C03650=1184.713,-44.316,-42.579,179.626,5.711,149.123
C03651=1184.719,-44.566,-42.567,179.624,5.710,149.123
C03652=1184.724,-44.815,-42.555,179.621,5.710,149.124
C03653=1184.729,-45.065,-42.544,179.619,5.709,149.125
C03654=1184.734,-45.315,-42.532,179.617,5.709,149.125
C03655=1184.740,-45.564,-42.520,179.614,5.709,149.126
C03656=1184.745,-45.814,-42.509,179.612,5.708,149.127
C03657=1184.750,-46.063,-42.496,179.609,5.708,149.127
C03658=1184.755,-46.313,-42.484,179.607,5.708,149.128
C03659=1184.761,-46.563,-42.473,179.605,5.708,149.129
C03660=1184.766,-46.813,-42.461,179.602,5.707,149.129
C03661=1184.771,-47.063,-42.449,179.600,5.707,149.130
C03662=1184.776,-47.312,-42.437,179.598,5.707,149.130
C03663=1184.781,-47.561,-42.425,179.595,5.706,149.131
C03664=1184.786,-47.811,-42.414,179.592,5.706,149.132
C03665=1184.791,-48.061,-42.402,179.591,5.706,149.132
C03666=1184.797,-48.310,-42.391,179.588,5.705,149.133
C03667=1184.802,-48.560,-42.379,179.586,5.705,149.134
C03668=1184.807,-48.810,-42.368,179.583,5.704,149.134
C03669=1184.812,-49.060,-42.356,179.581,5.704,149.135
C03670=1184.818,-49.330,-42.343,179.579,5.704,149.136
C03671=1184.824,-49.600,-42.330,179.576,5.704,149.136
C03672=1184.829,-49.871,-42.318,179.573,5.703,149.137
C03673=1184.835,-50.141,-42.305,179.571,5.703,149.138
C03674=1184.841,-50.390,-42.293,179.568,5.702,149.138
C03675=1184.845,-50.640,-42.282,179.566,5.702,149.139
C03676=1184.851,-50.890,-42.270,179.564,5.702,149.140
C03677=1184.855,-51.140,-42.259,179.561,5.701,149.140
C03678=1184.861,-51.389,-42.247,179.559,5.701,149.141
C03679=1184.866,-51.639,-42.235,179.557,5.701,149.142
C03680=1184.871,-51.889,-42.224,179.554,5.701,149.142
C03681=1184.877,-52.138,-42.212,179.552,5.700,149.143
C03682=1184.882,-52.388,-42.201,179.550,5.700,149.143
C03683=1184.887,-52.638,-42.189,179.547,5.700,149.144
C03684=1184.892,-52.887,-42.178,179.544,5.699,149.145
C03685=1184.897,-53.137,-42.166,179.542,5.698,149.145
C03686=1184.903,-53.386,-42.155,179.540,5.699,149.146
C03687=1184.908,-53.636,-42.143,179.538,5.698,149.147
C03688=1184.913,-53.886,-42.132,179.535,5.698,149.147
C03689=1184.918,-54.136,-42.120,179.533,5.697,149.148
C03690=1184.923,-54.385,-42.109,179.531,5.698,149.149
C03691=1184.928,-54.635,-42.097,179.528,5.697,149.149
C03692=1184.934,-54.884,-42.086,179.526,5.696,149.150
C03693=1184.939,-55.134,-42.074,179.524,5.697,149.150
C03694=1184.944,-55.384,-42.063,179.521,5.696,149.151
C03695=1184.949,-55.634,-42.051,179.519,5.695,149.152
C03696=1184.954,-55.883,-42.040,179.516,5.695,149.152
C03697=1184.960,-56.133,-42.028,179.514,5.695,149.153
C03698=1184.965,-56.382,-42.017,179.512,5.695,149.154
C03699=1184.970,-56.633,-42.006,179.509,5.694,149.154
C03700=1184.975,-56.882,-41.994,179.507,5.694,149.155
C03701=1184.981,-57.132,-41.983,179.505,5.694,149.155
C03702=1184.986,-57.381,-41.971,179.502,5.693,149.156
C03703=1184.990,-57.631,-41.960,179.500,5.694,149.157
C03704=1184.996,-57.881,-41.948,179.498,5.693,149.158
C03705=1185.001,-58.130,-41.937,179.495,5.692,149.158
C03706=1185.007,-58.380,-41.926,179.493,5.692,149.159
C03707=1185.012,-58.630,-41.915,179.491,5.692,149.159
C03708=1185.016,-58.880,-41.904,179.488,5.691,149.160
C03709=1185.022,-59.129,-41.892,179.486,5.691,149.161
C03710=1185.027,-59.378,-41.881,179.484,5.691,149.161
C03711=1185.033,-59.629,-41.870,179.482,5.691,149.162
C03712=1185.037,-59.879,-41.858,179.479,5.690,149.162
C03713=1185.043,-60.128,-41.847,179.477,5.691,149.163
C03714=1185.048,-60.378,-41.836,179.475,5.690,149.164
C03715=1185.053,-60.628,-41.825,179.472,5.689,149.164
C03716=1185.058,-60.878,-41.813,179.470,5.690,149.165
C03717=1185.064,-61.127,-41.802,179.467,5.689,149.166
C03718=1185.068,-61.376,-41.791,179.465,5.688,149.166
C03719=1185.074,-61.627,-41.780,179.462,5.688,149.167
C03720=1185.080,-61.876,-41.769,179.460,5.688,149.168
C03721=1185.084,-62.125,-41.757,179.458,5.688,149.168
C03722=1185.090,-62.375,-41.746,179.455,5.687,149.169
C03723=1185.095,-62.625,-41.735,179.453,5.688,149.170
C03724=1185.100,-62.874,-41.724,179.451,5.687,149.170
C03725=1185.105,-63.124,-41.712,179.448,5.686,149.171
C03726=1185.110,-63.375,-41.702,179.446,5.687,149.171
C03727=1185.116,-63.624,-41.691,179.444,5.686,149.172
C03728=1185.121,-63.873,-41.679,179.442,5.685,149.173
C03729=1185.126,-64.124,-41.668,179.439,5.686,149.173
C03730=1185.131,-64.373,-41.657,179.437,5.685,149.174
C03731=1185.137,-64.623,-41.645,179.435,5.685,149.175
C03732=1185.142,-64.873,-41.635,179.433,5.685,149.175
C03733=1185.147,-65.122,-41.624,179.430,5.684,149.176
C03734=1185.152,-65.371,-41.613,179.428,5.684,149.176
C03735=1185.158,-65.621,-41.602,179.426,5.684,149.177
C03736=1185.163,-65.871,-41.591,179.423,5.684,149.178
C03737=1185.168,-66.121,-41.580,179.421,5.683,149.178
C03738=1185.173,-66.370,-41.569,179.419,5.683,149.179
C03739=1185.179,-66.620,-41.557,179.416,5.683,149.180
C03740=1185.184,-66.870,-41.547,179.414,5.682,149.180
C03741=1185.189,-67.119,-41.536,179.412,5.682,149.181
C03742=1185.194,-67.369,-41.525,179.409,5.682,149.182
C03743=1185.199,-67.619,-41.513,179.407,5.681,149.182
C03744=1185.205,-67.869,-41.503,179.405,5.682,149.183
C03745=1185.210,-68.118,-41.492,179.402,5.681,149.183
C03746=1185.215,-68.367,-41.481,179.400,5.680,149.184
C03747=1185.221,-68.618,-41.470,179.398,5.681,149.185
C03748=1185.225,-68.868,-41.458,179.395,5.680,149.185
C03749=1185.231,-69.117,-41.448,179.393,5.680,149.186
C03750=1185.236,-69.367,-41.437,179.391,5.680,149.187
C03751=1185.241,-69.616,-41.427,179.388,5.680,149.187
C03752=1185.247,-69.866,-41.415,179.386,5.679,149.188
C03753=1185.252,-70.116,-41.404,179.384,5.679,149.188
C03754=1185.257,-70.365,-41.393,179.381,5.679,149.189
C03755=1185.262,-70.616,-41.383,179.379,5.678,149.190
C03756=1185.267,-70.865,-41.372,179.377,5.678,149.190
C03757=1185.272,-71.115,-41.361,179.374,5.678,149.191
C03758=1185.278,-71.365,-41.350,179.372,5.677,149.192
C03759=1185.283,-71.614,-41.339,179.370,5.677,149.192
C03760=1185.289,-71.864,-41.329,179.367,5.677,149.193
C03761=1185.293,-72.113,-41.318,179.366,5.677,149.193
C03762=1185.298,-72.364,-41.307,179.363,5.677,149.194
C03763=1185.304,-72.613,-41.296,179.360,5.676,149.195
C03764=1185.309,-72.863,-41.285,179.359,5.676,149.195
C03765=1185.315,-73.113,-41.275,179.356,5.676,149.196
C03766=1185.320,-73.362,-41.263,179.354,5.675,149.197
C03767=1185.325,-73.612,-41.253,179.352,5.675,149.197
C03768=1185.330,-73.862,-41.242,179.349,5.675,149.198
C03769=1185.336,-74.111,-41.232,179.347,5.674,149.199
C03770=1185.341,-74.361,-41.221,179.345,5.674,149.199
C03771=1185.346,-74.610,-41.210,179.342,5.674,149.200
C03772=1185.351,-74.860,-41.200,179.340,5.674,149.201
C03773=1185.357,-75.110,-41.189,179.338,5.674,149.201
C03774=1185.362,-75.381,-41.177,179.335,5.673,149.202
C03775=1185.368,-75.653,-41.166,179.333,5.673,149.202
C03776=1185.374,-75.923,-41.154,179.331,5.673,149.203
C03777=1185.379,-76.194,-41.143,179.328,5.673,149.204
C03778=1185.385,-76.443,-41.132,179.326,5.672,149.204
C03779=1185.390,-76.693,-41.121,179.323,5.672,149.205
C03780=1185.395,-76.943,-41.111,179.321,5.672,149.206
C03781=1185.400,-77.193,-41.100,179.319,5.671,149.206
C03782=1185.406,-77.442,-41.090,179.317,5.672,149.207
C03783=1185.411,-77.692,-41.079,179.314,5.671,149.208
C03784=1185.416,-77.942,-41.069,179.312,5.670,149.208
C03785=1185.422,-78.192,-41.057,179.310,5.671,149.209
C03786=1185.427,-78.441,-41.047,179.307,5.670,149.210
C03787=1185.432,-78.692,-41.036,179.305,5.669,149.210
C03788=1185.438,-78.941,-41.026,179.303,5.670,149.211
C03789=1185.443,-79.191,-41.015,179.300,5.669,149.211
C03790=1185.448,-79.440,-41.004,179.299,5.669,149.212
C03791=1185.453,-79.691,-40.994,179.296,5.669,149.213
C03792=1185.458,-79.940,-40.984,179.293,5.669,149.213
C03793=1185.463,-80.189,-40.973,179.292,5.669,149.214
C03794=1185.468,-80.439,-40.963,179.289,5.668,149.215
C03795=1185.474,-80.688,-40.953,179.287,5.668,149.215
C03796=1185.479,-80.939,-40.942,179.285,5.668,149.216
C03797=1185.485,-81.188,-40.932,179.282,5.667,149.216
C03798=1185.490,-81.439,-40.921,179.280,5.667,149.217
C03799=1185.495,-81.687,-40.910,179.278,5.667,149.218
C03800=1185.500,-81.938,-40.900,179.275,5.667,149.218
C03801=1185.505,-82.187,-40.889,179.274,5.667,149.219
C03802=1185.511,-82.437,-40.879,179.271,5.666,149.220
C03803=1185.516,-82.687,-40.869,179.269,5.667,149.220
C03804=1185.522,-82.937,-40.859,179.267,5.666,149.221
C03805=1185.527,-83.187,-40.848,179.264,5.665,149.221
C03806=1185.532,-83.436,-40.837,179.262,5.666,149.222
C03807=1185.537,-83.685,-40.827,179.260,5.665,149.223
C03808=1185.542,-83.936,-40.816,179.258,5.665,149.223
C03809=1185.547,-84.185,-40.807,179.255,5.665,149.224
C03810=1185.552,-84.435,-40.796,179.253,5.664,149.225
C03811=1185.558,-84.685,-40.786,179.251,5.665,149.225
C03812=1185.564,-84.934,-40.776,179.248,5.664,149.226
C03813=1185.569,-85.184,-40.765,179.246,5.664,149.226
C03814=1185.574,-85.434,-40.755,179.244,5.664,149.227
C03815=1185.579,-85.684,-40.744,179.241,5.663,149.228
C03816=1185.585,-85.934,-40.734,179.239,5.663,149.228
C03817=1185.590,-86.183,-40.724,179.237,5.663,149.229
C03818=1185.595,-86.433,-40.714,179.235,5.663,149.230
C03819=1185.600,-86.683,-40.704,179.232,5.663,149.230
C03820=1185.605,-86.932,-40.693,179.230,5.662,149.231
C03821=1185.610,-87.182,-40.682,179.228,5.662,149.231
C03822=1185.616,-87.431,-40.672,179.226,5.662,149.232
C03823=1185.621,-87.681,-40.662,179.224,5.662,149.233
C03824=1185.626,-87.931,-40.652,179.221,5.661,149.233
C03825=1185.632,-88.180,-40.642,179.220,5.661,149.234
C03826=1185.637,-88.431,-40.632,179.217,5.661,149.235
C03827=1185.642,-88.681,-40.621,179.214,5.660,149.235
C03828=1185.647,-88.930,-40.612,179.213,5.660,149.236
C03829=1185.653,-89.180,-40.602,179.210,5.660,149.236
C03830=1185.658,-89.430,-40.591,179.208,5.660,149.237
C03831=1185.663,-89.679,-40.581,179.206,5.660,149.238
C03832=1185.669,-89.929,-40.571,179.203,5.659,149.238
C03833=1185.673,-90.179,-40.561,179.202,5.659,149.239
C03834=1185.679,-90.428,-40.550,179.199,5.659,149.240
C03835=1185.685,-90.678,-40.540,179.197,5.659,149.240
C03836=1185.690,-90.928,-40.530,179.195,5.658,149.241
C03837=1185.694,-91.177,-40.520,179.192,5.659,149.241
C03838=1185.700,-91.427,-40.510,179.190,5.658,149.242
C03839=1185.705,-91.677,-40.499,179.188,5.658,149.243
C03840=1185.711,-91.927,-40.490,179.186,5.658,149.243
C03841=1185.716,-92.177,-40.480,179.183,5.657,149.244
C03842=1185.721,-92.426,-40.470,179.181,5.658,149.245
C03843=1185.726,-92.676,-40.459,179.179,5.657,149.245
C03844=1185.732,-92.926,-40.449,179.177,5.657,149.246
C03845=1185.737,-93.175,-40.440,179.174,5.657,149.246
C03846=1185.742,-93.425,-40.429,179.172,5.656,149.247
C03847=1185.748,-93.676,-40.420,179.170,5.656,149.248
C03848=1185.753,-93.925,-40.409,179.168,5.656,149.248
C03849=1185.758,-94.174,-40.400,179.166,5.656,149.249
C03850=1185.763,-94.425,-40.389,179.163,5.656,149.250
C03851=1185.769,-94.674,-40.379,179.162,5.656,149.250
C03852=1185.774,-94.923,-40.369,179.159,5.655,149.251
C03853=1185.780,-95.174,-40.360,179.157,5.655,149.251
C03854=1185.785,-95.424,-40.349,179.155,5.655,149.252
C03855=1185.789,-95.673,-40.340,179.152,5.655,149.253
C03856=1185.795,-95.923,-40.329,179.150,5.655,149.253
C03857=1185.801,-96.173,-40.320,179.148,5.654,149.254
C03858=1185.806,-96.422,-40.310,179.146,5.654,149.254
C03859=1185.811,-96.672,-40.300,179.143,5.654,149.255
C03860=1185.816,-96.922,-40.290,179.141,5.653,149.256
C03861=1185.822,-97.172,-40.281,179.139,5.653,149.256
C03862=1185.827,-97.421,-40.270,179.136,5.653,149.257
C03863=1185.832,-97.671,-40.260,179.135,5.653,149.257
C03864=1185.837,-97.921,-40.250,179.132,5.653,149.258
C03865=1185.843,-98.171,-40.241,179.130,5.653,149.259
C03866=1185.848,-98.420,-40.231,179.128,5.652,149.259
C03867=1185.853,-98.670,-40.221,179.126,5.653,149.260
C03868=1185.859,-98.920,-40.211,179.124,5.652,149.261
C03869=1185.864,-99.170,-40.201,179.121,5.651,149.261
C03870=1185.869,-99.419,-40.191,179.119,5.651,149.262
C03871=1185.875,-99.669,-40.182,179.117,5.651,149.262
C03872=1185.880,-99.919,-40.172,179.115,5.651,149.263
C03873=1185.885,-100.168,-40.162,179.112,5.651,149.264
C03874=1185.890,-100.419,-40.153,179.110,5.651,149.264
C03875=1185.896,-100.668,-40.142,179.108,5.650,149.265
C03876=1185.900,-100.917,-40.133,179.106,5.651,149.266
C03877=1185.906,-101.168,-40.123,179.103,5.650,149.266
C03878=1185.912,-101.439,-40.112,179.101,5.649,149.267
C03879=1185.918,-101.711,-40.102,179.099,5.650,149.267
C03880=1185.924,-101.982,-40.092,179.096,5.649,149.268
C03881=1185.929,-102.254,-40.081,179.094,5.649,149.269
C03882=1185.935,-102.504,-40.071,179.092,5.649,149.269
C03883=1185.939,-102.754,-40.061,179.089,5.649,149.270
C03884=1185.945,-103.003,-40.051,179.088,5.649,149.271
C03885=1185.950,-103.253,-40.042,179.085,5.648,149.271
C03886=1185.956,-103.503,-40.032,179.083,5.649,149.272
C03887=1185.961,-103.753,-40.023,179.081,5.648,149.272
C03888=1185.966,-104.002,-40.013,179.079,5.648,149.273
C03889=1185.972,-104.252,-40.004,179.077,5.648,149.274
C03890=1185.977,-104.501,-39.994,179.075,5.648,149.274
C03891=1185.982,-104.752,-39.985,179.072,5.647,149.275
C03892=1185.987,-105.002,-39.974,179.070,5.647,149.276
C03893=1185.992,-105.251,-39.965,179.068,5.647,149.276
C03894=1185.998,-105.501,-39.955,179.065,5.646,149.277
C03895=1186.003,-105.750,-39.946,179.063,5.647,149.277
C03896=1186.009,-106.000,-39.936,179.061,5.646,149.278
C03897=1186.014,-106.250,-39.926,179.059,5.646,149.279
C03898=1186.020,-106.500,-39.917,179.057,5.646,149.279
C03899=1186.024,-106.749,-39.907,179.055,5.646,149.280
C03900=1186.030,-107.000,-39.898,179.053,5.645,149.280
C03901=1186.035,-107.250,-39.889,179.050,5.646,149.281
C03902=1186.040,-107.499,-39.879,179.048,5.645,149.282
C03903=1186.046,-107.749,-39.870,179.046,5.645,149.282
C03904=1186.051,-107.998,-39.860,179.043,5.645,149.283
C03905=1186.056,-108.249,-39.850,179.042,5.645,149.283
C03906=1186.061,-108.498,-39.841,179.039,5.644,149.284
C03907=1186.067,-108.748,-39.831,179.038,5.644,149.285
C03908=1186.072,-108.997,-39.822,179.035,5.644,149.285
C03909=1186.077,-109.247,-39.813,179.033,5.643,149.286
C03910=1186.083,-109.497,-39.803,179.031,5.644,149.287
C03911=1186.088,-109.746,-39.794,179.028,5.643,149.287
C03912=1186.094,-109.997,-39.784,179.026,5.643,149.288
C03913=1186.099,-110.246,-39.775,179.024,5.643,149.288
C03914=1186.103,-110.496,-39.765,179.022,5.643,149.289
C03915=1186.109,-110.746,-39.756,179.019,5.643,149.290
C03916=1186.114,-110.996,-39.746,179.018,5.643,149.290
C03917=1186.120,-111.246,-39.737,179.015,5.642,149.291
C03918=1186.125,-111.496,-39.728,179.014,5.642,149.291
C03919=1186.130,-111.745,-39.718,179.011,5.642,149.292
C03920=1186.136,-111.995,-39.709,179.009,5.642,149.293
C03921=1186.141,-112.244,-39.699,179.007,5.641,149.293
C03922=1186.146,-112.494,-39.690,179.005,5.641,149.294
C03923=1186.152,-112.744,-39.681,179.002,5.641,149.295
C03924=1186.157,-112.994,-39.671,179.001,5.641,149.295
C03925=1186.162,-113.243,-39.662,178.998,5.641,149.296
C03926=1186.168,-113.494,-39.653,178.996,5.641,149.296
C03927=1186.173,-113.743,-39.644,178.994,5.640,149.297
C03928=1186.178,-113.993,-39.634,178.992,5.640,149.297
C03929=1186.184,-114.243,-39.625,178.989,5.640,149.298
C03930=1186.189,-114.493,-39.616,178.988,5.640,149.299
C03931=1186.194,-114.742,-39.606,178.985,5.640,149.299
C03932=1186.200,-114.992,-39.597,178.983,5.640,149.300
C03933=1186.205,-115.242,-39.588,178.981,5.639,149.301
C03934=1186.210,-115.492,-39.579,178.979,5.640,149.301
C03935=1186.215,-115.741,-39.569,178.977,5.639,149.302
C03936=1186.221,-115.991,-39.560,178.975,5.639,149.302
C03937=1186.226,-116.241,-39.551,178.972,5.638,149.303
C03938=1186.231,-116.491,-39.542,178.970,5.639,149.304
C03939=1186.237,-116.740,-39.532,178.968,5.638,149.304
C03940=1186.242,-116.990,-39.523,178.966,5.639,149.305
C03941=1186.248,-117.239,-39.514,178.964,5.638,149.305
C03942=1186.253,-117.489,-39.505,178.962,5.638,149.306
C03943=1186.259,-117.739,-39.496,178.960,5.637,149.307
C03944=1186.264,-117.989,-39.486,178.957,5.638,149.307
C03945=1186.269,-118.239,-39.477,178.955,5.637,149.308
C03946=1186.274,-118.488,-39.469,178.953,5.637,149.308
C03947=1186.280,-118.739,-39.459,178.951,5.637,149.309
C03948=1186.285,-118.988,-39.450,178.949,5.637,149.310
C03949=1186.290,-119.238,-39.441,178.947,5.636,149.310
C03950=1186.295,-119.487,-39.432,178.945,5.637,149.311
C03951=1186.300,-119.737,-39.423,178.942,5.636,149.311
C03952=1186.306,-119.988,-39.413,178.940,5.636,149.312
C03953=1186.311,-120.237,-39.404,178.938,5.636,149.313
C03954=1186.316,-120.487,-39.395,178.936,5.636,149.313
C03955=1186.322,-120.737,-39.387,178.934,5.635,149.314
C03956=1186.327,-120.987,-39.378,178.932,5.636,149.314
C03957=1186.333,-121.236,-39.369,178.930,5.635,149.315
C03958=1186.338,-121.486,-39.359,178.928,5.635,149.316
C03959=1186.343,-121.735,-39.350,178.925,5.634,149.316
C03960=1186.348,-121.985,-39.341,178.923,5.635,149.317
C03961=1186.354,-122.235,-39.332,178.921,5.634,149.317
C03962=1186.359,-122.485,-39.323,178.919,5.634,149.318
C03963=1186.365,-122.735,-39.314,178.917,5.634,149.319
C03964=1186.370,-122.985,-39.305,178.915,5.634,149.319
C03965=1186.375,-123.235,-39.296,178.912,5.633,149.320
C03966=1186.380,-123.485,-39.287,178.911,5.633,149.320
C03967=1186.386,-123.734,-39.279,178.908,5.633,149.321
C03968=1186.391,-123.984,-39.270,178.907,5.633,149.321
C03969=1186.396,-124.234,-39.261,178.905,5.633,149.322
C03970=1186.402,-124.484,-39.251,178.902,5.633,149.323
C03971=1186.407,-124.734,-39.242,178.900,5.633,149.323
C03972=1186.413,-124.983,-39.234,178.898,5.632,149.324
C03973=1186.418,-125.233,-39.225,178.896,5.633,149.325
C03974=1186.423,-125.482,-39.216,178.894,5.632,149.325
C03975=1186.429,-125.732,-39.207,178.892,5.632,149.326
C03976=1186.434,-125.982,-39.198,178.889,5.632,149.326
C03977=1186.439,-126.232,-39.189,178.887,5.632,149.327
C03978=1186.444,-126.482,-39.180,178.885,5.631,149.327
C03979=1186.450,-126.732,-39.171,178.883,5.632,149.328
C03980=1186.455,-126.982,-39.162,178.881,5.631,149.329
C03981=1186.461,-127.231,-39.154,178.879,5.631,149.329
C03982=1186.039,-127.242,-39.194,178.875,5.634,149.331
C03983=1186.034,-126.992,-39.202,178.877,5.634,149.331
C03984=1186.029,-126.742,-39.211,178.879,5.635,149.330
C03985=1186.023,-126.493,-39.219,178.881,5.634,149.329
C03986=1186.018,-126.243,-39.228,178.884,5.635,149.329
C03987=1186.013,-125.993,-39.237,178.886,5.635,149.328
C03988=1186.007,-125.743,-39.246,178.888,5.636,149.328
C03989=1186.002,-125.493,-39.255,178.890,5.635,149.327
C03990=1185.996,-125.243,-39.264,178.892,5.636,149.326
C03991=1185.991,-124.993,-39.273,178.894,5.636,149.326
C03992=1185.985,-124.744,-39.282,178.896,5.636,149.325
C03993=1185.980,-124.494,-39.291,178.898,5.636,149.324
C03994=1185.975,-124.245,-39.300,178.901,5.637,149.324
C03995=1185.970,-123.995,-39.308,178.902,5.637,149.324
C03996=1185.965,-123.745,-39.317,178.905,5.637,149.323
C03997=1185.959,-123.495,-39.326,178.906,5.637,149.322
C03998=1185.954,-123.245,-39.336,178.909,5.637,149.322
C03999=1185.948,-122.995,-39.345,178.911,5.637,149.321
C04000=1185.943,-122.746,-39.354,178.913,5.638,149.320
C04001=1185.938,-122.497,-39.363,178.915,5.638,149.320
C04002=1185.933,-122.247,-39.372,178.918,5.638,149.319
C04003=1185.927,-121.997,-39.381,178.919,5.638,149.319
C04004=1185.922,-121.747,-39.389,178.921,5.638,149.318
C04005=1185.916,-121.497,-39.399,178.924,5.638,149.317
C04006=1185.911,-121.247,-39.408,178.926,5.638,149.317
C04007=1185.906,-120.997,-39.417,178.928,5.639,149.316
C04008=1185.901,-120.747,-39.426,178.930,5.638,149.316
C04009=1185.896,-120.497,-39.435,178.932,5.639,149.315
C04010=1185.889,-120.248,-39.444,178.934,5.639,149.314
C04011=1185.884,-119.999,-39.453,178.936,5.640,149.314
C04012=1185.879,-119.749,-39.462,178.939,5.639,149.313
C04013=1185.874,-119.499,-39.471,178.941,5.640,149.313
C04014=1185.869,-119.249,-39.480,178.943,5.639,149.312
C04015=1185.863,-118.999,-39.489,178.945,5.640,149.311
C04016=1185.858,-118.749,-39.498,178.947,5.640,149.311
C04017=1185.853,-118.500,-39.508,178.949,5.641,149.310
C04018=1185.848,-118.250,-39.517,178.951,5.640,149.310
C04019=1185.842,-118.000,-39.526,178.954,5.641,149.309
C04020=1185.837,-117.750,-39.535,178.956,5.641,149.308
C04021=1185.832,-117.500,-39.544,178.958,5.641,149.308
C04022=1185.826,-117.250,-39.553,178.960,5.641,149.307
C04023=1185.822,-117.001,-39.563,178.962,5.642,149.307
C04024=1185.816,-116.751,-39.572,178.964,5.641,149.306
C04025=1185.810,-116.501,-39.581,178.966,5.642,149.305
C04026=1185.805,-116.251,-39.590,178.968,5.642,149.305
C04027=1185.800,-116.002,-39.600,178.971,5.642,149.304
C04028=1185.794,-115.753,-39.609,178.973,5.642,149.304
C04029=1185.789,-115.503,-39.618,178.975,5.643,149.303
C04030=1185.784,-115.253,-39.627,178.977,5.642,149.302
C04031=1185.778,-115.003,-39.636,178.979,5.643,149.302
C04032=1185.773,-114.754,-39.646,178.981,5.643,149.301
C04033=1185.768,-114.504,-39.655,178.984,5.644,149.301
C04034=1185.762,-114.254,-39.664,178.986,5.643,149.300
C04035=1185.757,-114.004,-39.674,178.988,5.644,149.299
C04036=1185.752,-113.754,-39.683,178.990,5.644,149.299
C04037=1185.746,-113.504,-39.692,178.992,5.644,149.298
C04038=1185.741,-113.254,-39.701,178.994,5.644,149.298
C04039=1185.736,-113.005,-39.711,178.996,5.645,149.297
C04040=1185.730,-112.755,-39.720,178.998,5.644,149.296
C04041=1185.725,-112.505,-39.729,179.001,5.645,149.296
C04042=1185.720,-112.256,-39.739,179.003,5.645,149.295
C04043=1185.714,-112.006,-39.748,179.005,5.645,149.295
C04044=1185.709,-111.756,-39.757,179.007,5.645,149.294
C04045=1185.704,-111.507,-39.767,179.009,5.646,149.293
C04046=1185.698,-111.257,-39.776,179.012,5.646,149.293
C04047=1185.693,-111.006,-39.785,179.014,5.646,149.292
C04048=1185.688,-110.756,-39.796,179.016,5.647,149.292
C04049=1185.683,-110.507,-39.804,179.018,5.646,149.291
C04050=1185.678,-110.257,-39.814,179.020,5.647,149.290
C04051=1185.672,-110.007,-39.824,179.022,5.647,149.290
C04052=1185.667,-109.757,-39.832,179.025,5.647,149.289
C04053=1185.662,-109.508,-39.842,179.027,5.647,149.288
C04054=1185.656,-109.258,-39.852,179.029,5.648,149.288
C04055=1185.651,-109.009,-39.861,179.031,5.647,149.287
C04056=1185.645,-108.759,-39.871,179.033,5.648,149.287
C04057=1185.640,-108.509,-39.880,179.035,5.648,149.286
C04058=1185.634,-108.259,-39.890,179.037,5.648,149.286
C04059=1185.629,-108.009,-39.899,179.040,5.648,149.285
C04060=1185.624,-107.760,-39.908,179.042,5.648,149.284
C04061=1185.619,-107.510,-39.918,179.044,5.648,149.284
C04062=1185.614,-107.261,-39.927,179.047,5.649,149.283
C04063=1185.608,-107.010,-39.937,179.048,5.649,149.282
C04064=1185.603,-106.761,-39.947,179.051,5.649,149.282
C04065=1185.598,-106.510,-39.956,179.052,5.649,149.281
C04066=1185.593,-106.261,-39.966,179.055,5.650,149.281
C04067=1185.587,-106.011,-39.975,179.057,5.650,149.280
C04068=1185.582,-105.762,-39.985,179.059,5.650,149.279
C04069=1185.577,-105.512,-39.994,179.062,5.651,149.279
C04070=1185.571,-105.262,-40.004,179.064,5.650,149.278
C04071=1185.566,-105.013,-40.013,179.066,5.651,149.277
C04072=1185.560,-104.763,-40.023,179.068,5.651,149.277
C04073=1185.556,-104.512,-40.033,179.071,5.651,149.276
C04074=1185.550,-104.263,-40.043,179.072,5.651,149.276
C04075=1185.545,-104.013,-40.052,179.075,5.651,149.275
C04076=1185.540,-103.764,-40.062,179.076,5.651,149.275
C04077=1185.534,-103.514,-40.071,179.079,5.652,149.274
C04078=1185.529,-103.264,-40.081,179.081,5.652,149.273
C04079=1185.524,-103.014,-40.090,179.083,5.652,149.273
C04080=1185.519,-102.764,-40.100,179.085,5.652,149.272
C04081=1185.514,-102.515,-40.110,179.088,5.653,149.271
C04082=1185.508,-102.265,-40.120,179.090,5.653,149.271
C04083=1185.503,-101.993,-40.130,179.092,5.653,149.270
C04084=1185.496,-101.722,-40.141,179.095,5.653,149.270
C04085=1185.490,-101.450,-40.151,179.097,5.654,149.269
C04086=1185.485,-101.179,-40.162,179.099,5.653,149.268
C04087=1185.479,-100.928,-40.172,179.102,5.654,149.268
C04088=1185.474,-100.679,-40.181,179.104,5.654,149.267
C04089=1185.469,-100.430,-40.191,179.106,5.654,149.266
C04090=1185.464,-100.179,-40.201,179.108,5.654,149.266
C04091=1185.459,-99.930,-40.211,179.111,5.655,149.265
C04092=1185.453,-99.680,-40.221,179.113,5.655,149.264
C04093=1185.448,-99.430,-40.230,179.115,5.655,149.264
C04094=1185.442,-99.181,-40.240,179.118,5.655,149.263
C04095=1185.437,-98.931,-40.250,179.119,5.655,149.263
C04096=1185.432,-98.681,-40.260,179.122,5.656,149.262
C04097=1185.426,-98.431,-40.270,179.123,5.656,149.261
C04098=1185.422,-98.182,-40.279,179.126,5.656,149.261
C04099=1185.416,-97.932,-40.289,179.128,5.656,149.260
C04100=1185.411,-97.682,-40.299,179.130,5.657,149.259
C04101=1185.406,-97.432,-40.309,179.133,5.657,149.259
C04102=1185.400,-97.182,-40.319,179.135,5.657,149.258
C04103=1185.395,-96.933,-40.328,179.137,5.657,149.258
C04104=1185.389,-96.683,-40.338,179.139,5.657,149.257
C04105=1185.384,-96.433,-40.349,179.142,5.658,149.256
C04106=1185.379,-96.183,-40.358,179.144,5.657,149.256
C04107=1185.374,-95.934,-40.368,179.146,5.658,149.255
C04108=1185.368,-95.684,-40.378,179.148,5.658,149.254
C04109=1185.363,-95.435,-40.388,179.150,5.658,149.254
C04110=1185.358,-95.185,-40.399,179.153,5.659,149.253
C04111=1185.352,-94.934,-40.408,179.154,5.659,149.253
C04112=1185.347,-94.685,-40.418,179.157,5.659,149.252
C04113=1185.342,-94.436,-40.428,179.159,5.659,149.251
C04114=1185.337,-94.185,-40.438,179.161,5.660,149.251
C04115=1185.331,-93.936,-40.449,179.163,5.659,149.250
C04116=1185.326,-93.686,-40.458,179.166,5.660,149.250
C04117=1185.321,-93.436,-40.468,179.168,5.660,149.249
C04118=1185.316,-93.186,-40.478,179.170,5.660,149.248
C04119=1185.311,-92.937,-40.488,179.173,5.661,149.248
C04120=1185.305,-92.687,-40.498,179.175,5.660,149.247
C04121=1185.300,-92.437,-40.509,179.177,5.661,149.247
C04122=1185.294,-92.187,-40.518,179.179,5.661,149.246
C04123=1185.289,-91.938,-40.528,179.182,5.661,149.245
C04124=1185.284,-91.688,-40.538,179.184,5.662,149.245
C04125=1185.279,-91.438,-40.549,179.186,5.662,149.244
C04126=1185.273,-91.188,-40.559,179.188,5.662,149.243
C04127=1185.268,-90.939,-40.568,179.190,5.662,149.243
C04128=1185.263,-90.689,-40.579,179.193,5.662,149.242
C04129=1185.258,-90.439,-40.589,179.195,5.663,149.242
C04130=1185.252,-90.190,-40.599,179.197,5.663,149.241
C04131=1185.247,-89.941,-40.609,179.200,5.663,149.240
C04132=1185.242,-89.690,-40.619,179.201,5.663,149.240
C04133=1185.236,-89.440,-40.629,179.204,5.664,149.239
C04134=1185.231,-89.191,-40.639,179.206,5.664,149.238
C04135=1185.226,-88.941,-40.649,179.208,5.664,149.238
C04136=1185.221,-88.691,-40.660,179.211,5.664,149.237
C04137=1185.215,-88.442,-40.670,179.213,5.664,149.237
C04138=1185.210,-88.191,-40.680,179.215,5.665,149.236
C04139=1185.205,-87.942,-40.691,179.217,5.665,149.235
C04140=1185.199,-87.692,-40.701,179.220,5.665,149.235
C04141=1185.195,-87.442,-40.711,179.222,5.666,149.234
C04142=1185.189,-87.193,-40.721,179.224,5.666,149.233
C04143=1185.184,-86.943,-40.731,179.226,5.666,149.233
C04144=1185.179,-86.693,-40.742,179.229,5.666,149.232
C04145=1185.173,-86.443,-40.752,179.231,5.666,149.232
C04146=1185.168,-86.193,-40.762,179.233,5.667,149.231
C04147=1185.163,-85.944,-40.772,179.235,5.667,149.230
C04148=1185.158,-85.694,-40.782,179.238,5.667,149.230
C04149=1185.153,-85.444,-40.793,179.240,5.667,149.229
C04150=1185.147,-85.195,-40.803,179.242,5.668,149.228
C04151=1185.141,-84.945,-40.813,179.245,5.668,149.228
C04152=1185.137,-84.696,-40.825,179.247,5.668,149.227
C04153=1185.131,-84.446,-40.835,179.249,5.668,149.227
C04154=1185.127,-84.196,-40.845,179.251,5.668,149.226
C04155=1185.121,-83.947,-40.855,179.253,5.669,149.225
C04156=1185.116,-83.697,-40.865,179.256,5.669,149.225
C04157=1185.111,-83.447,-40.876,179.258,5.669,149.224
C04158=1185.105,-83.197,-40.886,179.260,5.670,149.224
C04159=1185.100,-82.947,-40.897,179.262,5.669,149.223
C04160=1185.094,-82.697,-40.907,179.265,5.670,149.222
C04161=1185.089,-82.448,-40.917,179.267,5.671,149.222
C04162=1185.084,-82.198,-40.928,179.269,5.670,149.221
C04163=1185.079,-81.949,-40.938,179.271,5.671,149.220
C04164=1185.074,-81.698,-40.949,179.273,5.671,149.220
C04165=1185.068,-81.449,-40.959,179.276,5.671,149.219
C04166=1185.063,-81.199,-40.970,179.278,5.672,149.219
C04167=1185.058,-80.949,-40.979,179.280,5.671,149.218
C04168=1185.053,-80.700,-40.990,179.283,5.672,149.217
C04169=1185.048,-80.450,-41.001,179.285,5.672,149.217
C04170=1185.042,-80.201,-41.011,179.287,5.672,149.216
C04171=1185.037,-79.950,-41.022,179.290,5.673,149.215
C04172=1185.032,-79.701,-41.032,179.292,5.673,149.215
C04173=1185.027,-79.451,-41.043,179.294,5.673,149.214
C04174=1185.021,-79.202,-41.053,179.297,5.673,149.213
C04175=1185.016,-78.951,-41.064,179.299,5.673,149.213
C04176=1185.011,-78.702,-41.074,179.301,5.674,149.212
C04177=1185.005,-78.452,-41.084,179.303,5.674,149.212
C04178=1185.000,-78.203,-41.096,179.305,5.674,149.211
C04179=1184.995,-77.953,-41.106,179.308,5.675,149.210
C04180=1184.990,-77.703,-41.116,179.310,5.675,149.210
C04181=1184.985,-77.454,-41.127,179.312,5.675,149.209
C04182=1184.980,-77.204,-41.138,179.315,5.675,149.208
C04183=1184.974,-76.954,-41.148,179.317,5.675,149.208
C04184=1184.968,-76.704,-41.159,179.319,5.676,149.207
C04185=1184.963,-76.455,-41.170,179.321,5.676,149.206
C04186=1184.958,-76.205,-41.181,179.324,5.676,149.206
C04187=1184.952,-75.934,-41.191,179.326,5.677,149.205
C04188=1184.946,-75.663,-41.204,179.329,5.677,149.205
C04189=1184.941,-75.391,-41.215,179.331,5.677,149.204
C04190=1184.935,-75.121,-41.227,179.334,5.677,149.203
C04191=1184.930,-74.871,-41.237,179.336,5.678,149.203
C04192=1184.925,-74.622,-41.248,179.338,5.678,149.202
C04193=1184.920,-74.372,-41.259,179.341,5.678,149.201
C04194=1184.913,-74.122,-41.269,179.343,5.679,149.201
C04195=1184.909,-73.873,-41.281,179.345,5.678,149.200
C04196=1184.903,-73.623,-41.291,179.348,5.679,149.199
C04197=1184.898,-73.373,-41.302,179.350,5.680,149.199
C04198=1184.893,-73.123,-41.313,179.352,5.679,149.198
C04199=1184.888,-72.874,-41.323,179.355,5.680,149.197
C04200=1184.883,-72.624,-41.334,179.357,5.680,149.197
C04201=1184.878,-72.374,-41.344,179.359,5.680,149.196
C04202=1184.872,-72.124,-41.356,179.361,5.681,149.196
C04203=1184.867,-71.875,-41.367,179.363,5.681,149.195
C04204=1184.862,-71.625,-41.377,179.366,5.681,149.194
C04205=1184.856,-71.376,-41.388,179.368,5.681,149.194
C04206=1184.851,-71.125,-41.399,179.370,5.681,149.193
C04207=1184.846,-70.877,-41.410,179.373,5.682,149.192
C04208=1184.840,-70.626,-41.421,179.375,5.682,149.192
C04209=1184.836,-70.376,-41.432,179.377,5.682,149.191
C04210=1184.830,-70.127,-41.442,179.380,5.683,149.191
C04211=1184.825,-69.877,-41.454,179.382,5.683,149.190
C04212=1184.820,-69.628,-41.464,179.384,5.683,149.189
C04213=1184.815,-69.378,-41.475,179.387,5.683,149.189
C04214=1184.809,-69.128,-41.486,179.389,5.684,149.188
C04215=1184.804,-68.879,-41.497,179.391,5.684,149.187
C04216=1184.799,-68.628,-41.508,179.393,5.684,149.187
C04217=1184.794,-68.379,-41.519,179.396,5.685,149.186
C04218=1184.788,-68.129,-41.530,179.398,5.685,149.186
C04219=1184.783,-67.880,-41.541,179.400,5.685,149.185
C04220=1184.778,-67.630,-41.551,179.403,5.686,149.184
C04221=1184.773,-67.380,-41.563,179.405,5.686,149.184
C04222=1184.767,-67.131,-41.573,179.407,5.686,149.183
C04223=1184.762,-66.881,-41.585,179.410,5.686,149.182
C04224=1184.757,-66.631,-41.596,179.412,5.686,149.182
C04225=1184.752,-66.381,-41.606,179.414,5.687,149.181
C04226=1184.747,-66.132,-41.617,179.417,5.687,149.180
C04227=1184.741,-65.882,-41.628,179.419,5.687,149.180
C04228=1184.736,-65.632,-41.640,179.421,5.688,149.179
C04229=1184.731,-65.383,-41.651,179.424,5.688,149.178
C04230=1184.725,-65.133,-41.662,179.425,5.688,149.178
C04231=1184.720,-64.883,-41.673,179.428,5.689,149.177
C04232=1184.715,-64.633,-41.683,179.431,5.689,149.177
C04233=1184.710,-64.384,-41.694,179.432,5.689,149.176
C04234=1184.704,-64.134,-41.706,179.435,5.689,149.175
C04235=1184.699,-63.884,-41.717,179.438,5.690,149.175
C04236=1184.694,-63.635,-41.728,179.440,5.689,149.174
C04237=1184.689,-63.385,-41.740,179.442,5.690,149.174
C04238=1184.684,-63.135,-41.750,179.445,5.691,149.173
C04239=1184.678,-62.886,-41.761,179.447,5.690,149.172
C04240=1184.673,-62.636,-41.773,179.449,5.691,149.172
C04241=1184.668,-62.386,-41.784,179.452,5.692,149.171
C04242=1184.663,-62.137,-41.795,179.454,5.691,149.170
C04243=1184.657,-61.887,-41.806,179.456,5.692,149.170
C04244=1184.653,-61.637,-41.818,179.459,5.692,149.169
C04245=1184.648,-61.387,-41.828,179.461,5.693,149.168
C04246=1184.642,-61.138,-41.840,179.463,5.693,149.168
C04247=1184.637,-60.888,-41.851,179.465,5.693,149.167
C04248=1184.632,-60.638,-41.862,179.468,5.694,149.166
C04249=1184.626,-60.389,-41.873,179.470,5.694,149.166
C04250=1184.621,-60.139,-41.885,179.472,5.694,149.165
C04251=1184.616,-59.889,-41.896,179.475,5.695,149.165
C04252=1184.611,-59.639,-41.908,179.477,5.695,149.164
C04253=1184.605,-59.390,-41.918,179.479,5.695,149.163
C04254=1184.600,-59.140,-41.930,179.482,5.695,149.163
C04255=1184.595,-58.890,-41.941,179.484,5.695,149.162
C04256=1184.591,-58.641,-41.952,179.486,5.696,149.161
C04257=1184.585,-58.391,-41.964,179.489,5.696,149.161
C04258=1184.580,-58.141,-41.974,179.492,5.697,149.160
C04259=1184.574,-57.891,-41.986,179.493,5.697,149.160
C04260=1184.570,-57.642,-41.998,179.496,5.697,149.159
C04261=1184.563,-57.392,-42.009,179.499,5.698,149.158
C04262=1184.559,-57.143,-42.020,179.500,5.698,149.158
C04263=1184.554,-56.893,-42.032,179.503,5.698,149.157
C04264=1184.549,-56.643,-42.044,179.505,5.698,149.156
C04265=1184.543,-56.394,-42.054,179.507,5.698,149.156
C04266=1184.538,-56.144,-42.066,179.510,5.699,149.155
C04267=1184.533,-55.894,-42.077,179.512,5.699,149.154
C04268=1184.528,-55.644,-42.089,179.515,5.700,149.154
C04269=1184.523,-55.395,-42.100,179.517,5.700,149.153
C04270=1184.517,-55.145,-42.112,179.519,5.700,149.153
C04271=1184.512,-54.896,-42.123,179.522,5.701,149.152
C04272=1184.507,-54.646,-42.135,179.524,5.701,149.151
C04273=1184.502,-54.396,-42.146,179.526,5.701,149.151
C04274=1184.497,-54.146,-42.158,179.529,5.701,149.150
C04275=1184.491,-53.897,-42.169,179.531,5.702,149.149
C04276=1184.486,-53.647,-42.181,179.533,5.702,149.149
C04277=1184.481,-53.397,-42.191,179.536,5.702,149.148
C04278=1184.475,-53.147,-42.203,179.538,5.703,149.147
C04279=1184.471,-52.897,-42.215,179.540,5.703,149.147
C04280=1184.465,-52.648,-42.226,179.543,5.703,149.146
C04281=1184.460,-52.399,-42.237,179.545,5.704,149.145
C04282=1184.455,-52.149,-42.249,179.548,5.704,149.145
C04283=1184.450,-51.899,-42.261,179.550,5.704,149.144
C04284=1184.444,-51.649,-42.272,179.552,5.704,149.144
C04285=1184.440,-51.399,-42.284,179.555,5.705,149.143
C04286=1184.434,-51.150,-42.295,179.557,5.706,149.142
C04287=1184.428,-50.900,-42.307,179.559,5.705,149.142
C04288=1184.424,-50.651,-42.319,179.562,5.706,149.141
C04289=1184.418,-50.401,-42.331,179.564,5.707,149.141
C04290=1184.414,-50.152,-42.342,179.566,5.706,149.140
C04291=1184.408,-49.881,-42.355,179.569,5.707,149.139
C04292=1184.402,-49.611,-42.367,179.572,5.707,149.138
C04293=1184.397,-49.341,-42.380,179.574,5.708,149.138
C04294=1184.391,-49.070,-42.392,179.577,5.708,149.137
C04295=1184.386,-48.821,-42.405,179.579,5.709,149.137
C04296=1184.380,-48.571,-42.417,179.581,5.708,149.136
C04297=1184.375,-48.322,-42.428,179.584,5.709,149.135
C04298=1184.370,-48.072,-42.440,179.586,5.710,149.135
C04299=1184.365,-47.822,-42.451,179.589,5.710,149.134
C04300=1184.360,-47.572,-42.463,179.591,5.710,149.133
C04301=1184.354,-47.322,-42.475,179.593,5.710,149.133
C04302=1184.349,-47.073,-42.486,179.596,5.711,149.132
C04303=1184.344,-46.824,-42.498,179.598,5.711,149.131
C04304=1184.339,-46.574,-42.510,179.600,5.711,149.131
C04305=1184.334,-46.324,-42.521,179.602,5.712,149.130
C04306=1184.329,-46.074,-42.533,179.605,5.712,149.129
C04307=1184.323,-45.825,-42.545,179.608,5.713,149.129
C04308=1184.318,-45.575,-42.557,179.610,5.712,149.128
C04309=1184.313,-45.326,-42.569,179.612,5.713,149.128
C04310=1184.308,-45.076,-42.581,179.615,5.714,149.127
C04311=1184.302,-44.826,-42.593,179.617,5.714,149.126
C04312=1184.298,-44.576,-42.604,179.619,5.714,149.126
C04313=1184.293,-44.327,-42.617,179.622,5.715,149.125
C04314=1184.287,-44.077,-42.629,179.624,5.715,149.124
C04315=1184.282,-43.827,-42.640,179.626,5.716,149.124
C04316=1184.276,-43.578,-42.651,179.629,5.716,149.123
C04317=1184.271,-43.329,-42.664,179.631,5.716,149.122
C04318=1184.266,-43.079,-42.676,179.634,5.716,149.122
C04319=1184.261,-42.829,-42.687,179.636,5.717,149.121
C04320=1184.256,-42.579,-42.699,179.639,5.718,149.121
C04321=1184.251,-42.330,-42.712,179.641,5.717,149.120
C04322=1184.245,-42.080,-42.724,179.643,5.718,149.119
C04323=1184.241,-41.830,-42.735,179.646,5.718,149.119
C04324=1184.235,-41.581,-42.748,179.648,5.719,149.118
C04325=1184.230,-41.331,-42.759,179.650,5.719,149.117
C04326=1184.225,-41.081,-42.771,179.653,5.719,149.117
C04327=1184.219,-40.832,-42.784,179.655,5.720,149.116
C04328=1184.215,-40.582,-42.795,179.658,5.720,149.115
C04329=1184.209,-40.332,-42.807,179.660,5.721,149.115
C04330=1184.204,-40.083,-42.820,179.662,5.721,149.114
C04331=1184.199,-39.833,-42.832,179.665,5.721,149.114
C04332=1184.193,-39.583,-42.843,179.668,5.722,149.113
C04333=1184.189,-39.334,-42.855,179.670,5.722,149.112
C04334=1184.184,-39.084,-42.867,179.672,5.722,149.112
C04335=1184.178,-38.834,-42.879,179.674,5.723,149.111
C04336=1184.173,-38.585,-42.892,179.677,5.723,149.111
C04337=1184.168,-38.335,-42.904,179.679,5.724,149.110
C04338=1184.162,-38.086,-42.916,179.682,5.724,149.109
C04339=1184.157,-37.836,-42.928,179.684,5.724,149.108
C04340=1184.153,-37.587,-42.940,179.686,5.725,149.108
C04341=1184.147,-37.337,-42.952,179.689,5.725,149.107
C04342=1184.142,-37.087,-42.964,179.692,5.726,149.107
C04343=1184.137,-36.837,-42.977,179.693,5.726,149.106
C04344=1184.132,-36.587,-42.989,179.696,5.726,149.105
C04345=1184.127,-36.337,-43.001,179.698,5.726,149.105
C04346=1184.121,-36.088,-43.013,179.701,5.727,149.104
C04347=1184.116,-35.838,-43.026,179.703,5.728,149.103
C04348=1184.111,-35.588,-43.038,179.705,5.727,149.103
C04349=1184.106,-35.339,-43.050,179.708,5.728,149.102
C04350=1184.101,-35.089,-43.062,179.711,5.728,149.101
C04351=1184.096,-34.840,-43.074,179.713,5.729,149.101
C04352=1184.090,-34.590,-43.086,179.716,5.730,149.100
C04353=1184.085,-34.341,-43.099,179.718,5.729,149.100
C04354=1184.080,-34.091,-43.111,179.720,5.730,149.099
C04355=1184.075,-33.841,-43.123,179.722,5.730,149.098
C04356=1184.069,-33.592,-43.135,179.725,5.731,149.098
C04357=1184.065,-33.342,-43.148,179.728,5.731,149.097
C04358=1184.060,-33.092,-43.161,179.729,5.731,149.096
C04359=1184.054,-32.842,-43.173,179.732,5.732,149.096
C04360=1184.049,-32.593,-43.185,179.735,5.732,149.095
C04361=1184.044,-32.343,-43.197,179.737,5.733,149.095
C04362=1184.038,-32.094,-43.210,179.740,5.734,149.094
C04363=1184.033,-31.844,-43.222,179.742,5.734,149.093
C04364=1184.028,-31.594,-43.234,179.744,5.734,149.093
C04365=1184.023,-31.345,-43.247,179.746,5.734,149.092
C04366=1184.018,-31.094,-43.259,179.749,5.735,149.091
C04367=1184.013,-30.845,-43.272,179.752,5.735,149.091
C04368=1184.008,-30.596,-43.284,179.754,5.736,149.090
C04369=1184.002,-30.346,-43.296,179.756,5.736,149.089
C04370=1183.997,-30.097,-43.309,179.759,5.736,149.089
C04371=1183.992,-29.847,-43.321,179.761,5.737,149.088
C04372=1183.987,-29.597,-43.333,179.763,5.738,149.088
C04373=1183.982,-29.347,-43.346,179.766,5.738,149.087
C04374=1183.977,-29.098,-43.359,179.769,5.738,149.086
C04375=1183.972,-28.848,-43.371,179.770,5.738,149.086
C04376=1183.966,-28.599,-43.383,179.773,5.739,149.085
C04377=1183.961,-28.349,-43.396,179.776,5.739,149.084
C04378=1183.956,-28.100,-43.408,179.778,5.740,149.084
C04379=1183.951,-27.849,-43.421,179.781,5.741,149.083
C04380=1183.946,-27.600,-43.433,179.783,5.741,149.083
C04381=1183.941,-27.351,-43.446,179.785,5.741,149.082
C04382=1183.936,-27.102,-43.458,179.788,5.741,149.081
C04383=1183.930,-26.851,-43.471,179.790,5.742,149.081
C04384=1183.925,-26.601,-43.484,179.793,5.742,149.080
C04385=1183.920,-26.352,-43.497,179.795,5.743,149.079
C04386=1183.915,-26.103,-43.509,179.798,5.744,149.079
C04387=1183.910,-25.853,-43.522,179.800,5.743,149.078
C04388=1183.904,-25.603,-43.534,179.802,5.744,149.077
C04389=1183.900,-25.353,-43.547,179.805,5.744,149.077
C04390=1183.895,-25.104,-43.559,179.807,5.745,149.076
C04391=1183.890,-24.855,-43.572,179.810,5.746,149.076
C04392=1183.884,-24.605,-43.585,179.813,5.746,149.075
C04393=1183.879,-24.354,-43.597,179.814,5.746,149.074
C04394=1183.874,-24.105,-43.610,179.817,5.747,149.074
C04395=1183.869,-23.835,-43.624,179.819,5.747,149.073
C04396=1183.863,-23.566,-43.637,179.822,5.747,149.072
C04397=1183.858,-23.296,-43.651,179.825,5.748,149.072
C04398=1183.852,-23.026,-43.665,179.827,5.748,149.071
C04399=1183.847,-22.777,-43.678,179.830,5.749,149.070
C04400=1183.842,-22.528,-43.691,179.832,5.750,149.070
C04401=1183.836,-22.278,-43.702,179.835,5.750,149.069
C04402=1183.832,-22.028,-43.715,179.838,5.751,149.068
C04403=1183.826,-21.778,-43.729,179.840,5.751,149.068
C04404=1183.821,-21.529,-43.741,179.842,5.751,149.067
C04405=1183.815,-21.279,-43.754,179.844,5.751,149.066
C04406=1183.811,-21.029,-43.767,179.847,5.752,149.066
C04407=1183.805,-20.780,-43.780,179.849,5.753,149.065
C04408=1183.800,-20.530,-43.793,179.852,5.753,149.065
C04409=1183.795,-20.281,-43.805,179.855,5.754,149.064
C04410=1183.790,-20.031,-43.818,179.857,5.754,149.063
C04411=1183.784,-19.782,-43.831,179.859,5.754,149.063
C04412=1183.779,-19.532,-43.844,179.862,5.755,149.062
C04413=1183.775,-19.282,-43.857,179.864,5.755,149.061
C04414=1183.770,-19.033,-43.870,179.867,5.756,149.061
C04415=1183.764,-18.783,-43.883,179.869,5.756,149.060
C04416=1183.759,-18.533,-43.896,179.872,5.757,149.060
C04417=1183.754,-18.284,-43.908,179.874,5.757,149.059
C04418=1183.749,-18.035,-43.921,179.877,5.758,149.058
C04419=1183.744,-17.784,-43.934,179.879,5.758,149.058
C04420=1183.739,-17.535,-43.947,179.881,5.758,149.057
C04421=1183.734,-17.286,-43.960,179.884,5.759,149.056
C04422=1183.728,-17.035,-43.973,179.886,5.760,149.056
C04423=1183.723,-16.786,-43.986,179.889,5.760,149.055
C04424=1183.718,-16.537,-43.998,179.891,5.760,149.054
C04425=1183.713,-16.287,-44.013,179.894,5.761,149.054
C04426=1183.708,-16.038,-44.025,179.896,5.762,149.053
C04427=1183.703,-15.788,-44.038,179.899,5.762,149.053
C04428=1183.698,-15.538,-44.051,179.901,5.762,149.052
C04429=1183.692,-15.289,-44.064,179.903,5.763,149.051
C04430=1183.687,-15.039,-44.077,179.906,5.763,149.051
C04431=1183.682,-14.789,-44.090,179.908,5.764,149.050
C04432=1183.677,-14.540,-44.103,179.911,5.764,149.049
C04433=1183.672,-14.290,-44.117,179.913,5.765,149.049
C04434=1183.667,-14.041,-44.130,179.916,5.765,149.048
C04435=1183.662,-13.791,-44.142,179.919,5.766,149.047
C04436=1183.656,-13.541,-44.156,179.921,5.767,149.047
C04437=1183.651,-13.292,-44.168,179.923,5.766,149.046
C04438=1183.647,-13.042,-44.181,179.926,5.767,149.046
C04439=1183.641,-12.793,-44.195,179.928,5.767,149.045
C04440=1183.636,-12.543,-44.208,179.930,5.768,149.044
C04441=1183.631,-12.293,-44.222,179.933,5.769,149.044
C04442=1183.626,-12.044,-44.234,179.936,5.769,149.043
C04443=1183.621,-11.794,-44.248,179.938,5.770,149.043
C04444=1183.616,-11.545,-44.261,179.940,5.770,149.042
C04445=1183.611,-11.295,-44.274,179.943,5.771,149.041
C04446=1183.605,-11.045,-44.287,179.946,5.771,149.041
C04447=1183.600,-10.796,-44.300,179.948,5.772,149.040
C04448=1183.595,-10.546,-44.314,179.950,5.772,149.039
C04449=1183.590,-10.297,-44.327,179.953,5.772,149.039
C04450=1183.585,-10.046,-44.340,179.955,5.773,149.038
C04451=1183.580,-9.798,-44.354,179.958,5.774,149.038
C04452=1183.575,-9.547,-44.367,179.960,5.774,149.037
C04453=1183.570,-9.298,-44.380,179.963,5.774,149.036
C04454=1183.565,-9.048,-44.394,179.965,5.775,149.036
C04455=1183.560,-8.799,-44.407,179.968,5.776,149.035
C04456=1183.554,-8.549,-44.420,179.970,5.776,149.034
C04457=1183.549,-8.300,-44.433,179.972,5.777,149.034
C04458=1183.544,-8.050,-44.447,179.975,5.778,149.033
C04459=1183.539,-7.800,-44.460,179.978,5.778,149.032
C04460=1183.534,-7.551,-44.473,179.980,5.778,149.032
C04461=1183.529,-7.301,-44.486,179.982,5.779,149.031
C04462=1183.523,-7.052,-44.500,179.985,5.779,149.031
C04463=1183.519,-6.802,-44.513,179.987,5.779,149.030
C04464=1183.513,-6.553,-44.527,179.990,5.780,149.029
C04465=1183.509,-6.303,-44.540,179.992,5.781,149.029
C04466=1183.503,-6.054,-44.553,179.995,5.781,149.028
C04467=1183.498,-5.804,-44.568,179.998,5.782,149.027
C04468=1183.493,-5.555,-44.580,180.000,5.783,149.027
C04469=1183.488,-5.305,-44.595,-179.998,5.783,149.026
C04470=1183.483,-5.056,-44.607,-179.995,5.783,149.026
C04471=1183.478,-4.806,-44.621,-179.992,5.784,149.025
C04472=1183.473,-4.556,-44.634,-179.990,5.785,149.024
C04473=1183.467,-4.306,-44.648,-179.988,5.785,149.024
C04474=1183.463,-4.056,-44.662,-179.985,5.786,149.023
C04475=1183.457,-3.807,-44.674,-179.983,5.787,149.023
C04476=1183.452,-3.557,-44.689,-179.980,5.787,149.022
C04477=1183.447,-3.308,-44.702,-179.978,5.787,149.021
C04478=1183.442,-3.058,-44.716,-179.975,5.787,149.020
C04479=1183.437,-2.809,-44.730,-179.973,5.788,149.020
C04480=1183.432,-2.559,-44.743,-179.971,5.789,149.019
C04481=1183.427,-2.310,-44.756,-179.968,5.789,149.019
C04482=1183.421,-2.060,-44.770,-179.966,5.790,149.018
C04483=1183.417,-1.811,-44.784,-179.963,5.790,149.017
C04484=1183.411,-1.561,-44.797,-179.960,5.791,149.017
C04485=1183.406,-1.311,-44.811,-179.958,5.791,149.016
C04486=1183.401,-1.062,-44.824,-179.956,5.792,149.016
C04487=1183.396,-0.812,-44.838,-179.953,5.793,149.015
C04488=1183.391,-0.563,-44.852,-179.950,5.793,149.014
C04489=1183.386,-0.313,-44.866,-179.948,5.794,149.014
C04490=1183.381,-0.064,-44.879,-179.945,5.794,149.013
C04491=1183.375,0.186,-44.892,-179.943,5.795,149.012
C04492=1183.371,0.436,-44.907,-179.941,5.796,149.012
C04493=1183.366,0.685,-44.920,-179.938,5.796,149.011
C04494=1183.360,0.935,-44.934,-179.935,5.797,149.011
C04495=1183.355,1.185,-44.948,-179.933,5.797,149.010
C04496=1183.350,1.434,-44.962,-179.930,5.798,149.009
C04497=1183.345,1.684,-44.975,-179.928,5.798,149.009
C04498=1183.340,1.933,-44.989,-179.925,5.799,149.008
C04499=1183.334,2.202,-45.004,-179.923,5.799,149.007
C04500=1183.329,2.471,-45.019,-179.920,5.800,149.007
C04501=1183.324,2.741,-45.034,-179.917,5.800,149.006
C04502=1183.318,3.010,-45.049,-179.915,5.801,149.006
C04503=1183.313,3.259,-45.062,-179.912,5.802,149.005
C04504=1183.308,3.509,-45.076,-179.910,5.802,149.004
C04505=1183.303,3.759,-45.090,-179.907,5.803,149.003
C04506=1183.298,4.008,-45.104,-179.905,5.803,149.003
C04507=1183.293,4.258,-45.118,-179.902,5.804,149.002
C04508=1183.288,4.507,-45.132,-179.900,5.804,149.002
C04509=1183.283,4.757,-45.145,-179.897,5.805,149.001
C04510=1183.278,5.006,-45.159,-179.895,5.806,149.000
C04511=1183.273,5.256,-45.173,-179.892,5.806,149.000
C04512=1183.267,5.505,-45.187,-179.889,5.807,148.999
C04513=1183.262,5.755,-45.202,-179.887,5.808,148.999
C04514=1183.258,6.005,-45.215,-179.885,5.808,148.998
C04515=1183.253,6.255,-45.229,-179.882,5.808,148.997
C04516=1183.247,6.504,-45.243,-179.880,5.809,148.997
C04517=1183.242,6.753,-45.257,-179.877,5.810,148.996
C04518=1183.237,7.003,-45.271,-179.875,5.810,148.995
C04519=1183.232,7.252,-45.285,-179.872,5.811,148.995
C04520=1183.227,7.502,-45.299,-179.870,5.812,148.994
C04521=1183.222,7.752,-45.312,-179.867,5.812,148.994
C04522=1183.217,8.001,-45.326,-179.864,5.813,148.993
C04523=1183.212,8.250,-45.341,-179.862,5.813,148.992
C04524=1183.207,8.500,-45.355,-179.860,5.814,148.992
C04525=1183.202,8.750,-45.369,-179.857,5.814,148.991
C04526=1183.196,8.999,-45.383,-179.855,5.815,148.991
C04527=1183.191,9.249,-45.397,-179.852,5.816,148.990
C04528=1183.186,9.498,-45.412,-179.849,5.816,148.989
C04529=1183.181,9.748,-45.426,-179.847,5.817,148.989
C04530=1183.176,9.997,-45.440,-179.845,5.818,148.988
C04531=1183.171,10.247,-45.454,-179.842,5.818,148.987
C04532=1183.166,10.496,-45.468,-179.839,5.819,148.987
C04533=1183.162,10.746,-45.482,-179.837,5.819,148.986
C04534=1183.156,10.995,-45.496,-179.835,5.820,148.986
C04535=1183.151,11.245,-45.510,-179.832,5.820,148.985
C04536=1183.146,11.494,-45.524,-179.830,5.821,148.984
C04537=1183.141,11.744,-45.539,-179.827,5.822,148.984
C04538=1183.136,11.994,-45.553,-179.824,5.822,148.983
C04539=1183.131,12.243,-45.567,-179.822,5.823,148.983
C04540=1183.126,12.492,-45.581,-179.819,5.824,148.982
C04541=1183.121,12.742,-45.596,-179.816,5.825,148.981
C04542=1183.116,12.992,-45.610,-179.814,5.826,148.981
C04543=1183.111,13.242,-45.624,-179.812,5.826,148.980
C04544=1183.105,13.491,-45.638,-179.809,5.827,148.979
C04545=1183.100,13.740,-45.652,-179.806,5.827,148.979
C04546=1183.095,13.990,-45.667,-179.804,5.828,148.978
C04547=1183.090,14.240,-45.681,-179.801,5.828,148.978
C04548=1183.085,14.490,-45.696,-179.799,5.829,148.977
C04549=1183.079,14.739,-45.710,-179.797,5.830,148.976
C04550=1183.074,14.988,-45.724,-179.794,5.830,148.976
C04551=1183.070,15.238,-45.739,-179.791,5.831,148.975
C04552=1183.065,15.487,-45.753,-179.789,5.832,148.975
C04553=1183.060,15.737,-45.767,-179.786,5.832,148.974
C04554=1183.055,15.987,-45.782,-179.784,5.833,148.973
C04555=1183.050,16.236,-45.796,-179.782,5.833,148.973
C04556=1183.044,16.485,-45.810,-179.779,5.834,148.972
C04557=1183.040,16.734,-45.825,-179.776,5.834,148.971
C04558=1183.035,16.984,-45.839,-179.774,5.835,148.971
C04559=1183.030,17.234,-45.853,-179.772,5.836,148.970
C04560=1183.025,17.484,-45.868,-179.769,5.836,148.970
C04561=1183.019,17.734,-45.883,-179.766,5.837,148.969
C04562=1183.014,17.983,-45.898,-179.764,5.838,148.969
C04563=1183.009,18.232,-45.912,-179.761,5.839,148.968
C04564=1183.004,18.481,-45.926,-179.758,5.839,148.967
C04565=1182.999,18.731,-45.940,-179.756,5.840,148.967
C04566=1182.994,18.981,-45.954,-179.753,5.841,148.966
C04567=1182.989,19.230,-45.969,-179.751,5.841,148.965
C04568=1182.984,19.480,-45.984,-179.749,5.842,148.965
C04569=1182.979,19.730,-45.998,-179.746,5.843,148.964
C04570=1182.974,19.979,-46.013,-179.743,5.843,148.964
C04571=1182.969,20.228,-46.028,-179.741,5.844,148.963
C04572=1182.964,20.478,-46.042,-179.739,5.844,148.962
C04573=1182.958,20.728,-46.057,-179.736,5.845,148.962
C04574=1182.954,20.977,-46.072,-179.734,5.846,148.961
C04575=1182.948,21.226,-46.086,-179.731,5.846,148.961
C04576=1182.943,21.476,-46.100,-179.728,5.848,148.960
C04577=1182.939,21.725,-46.115,-179.725,5.848,148.959
C04578=1182.933,21.975,-46.130,-179.723,5.849,148.959
C04579=1182.928,22.224,-46.145,-179.720,5.849,148.958
C04580=1182.923,22.474,-46.159,-179.718,5.850,148.957
C04581=1182.918,22.724,-46.173,-179.716,5.851,148.957
C04582=1182.913,22.973,-46.189,-179.713,5.851,148.956
C04583=1182.908,23.223,-46.203,-179.710,5.852,148.956
C04584=1182.903,23.472,-46.218,-179.708,5.853,148.955
C04585=1182.898,23.722,-46.233,-179.705,5.853,148.954
C04586=1182.893,23.972,-46.247,-179.703,5.854,148.954
C04587=1182.888,24.221,-46.262,-179.701,5.854,148.953
C04588=1182.883,24.470,-46.277,-179.697,5.856,148.953
C04589=1182.878,24.719,-46.292,-179.695,5.856,148.952
C04590=1182.873,24.970,-46.307,-179.693,5.857,148.952
C04591=1182.868,25.219,-46.322,-179.690,5.858,148.951
C04592=1182.863,25.468,-46.336,-179.687,5.858,148.950
C04593=1182.858,25.718,-46.351,-179.685,5.859,148.950
C04594=1182.853,25.967,-46.366,-179.682,5.859,148.949
C04595=1182.848,26.217,-46.381,-179.680,5.860,148.948
C04596=1182.842,26.467,-46.396,-179.678,5.861,148.948
C04597=1182.838,26.716,-46.411,-179.674,5.862,148.947
C04598=1182.833,26.965,-46.425,-179.672,5.863,148.947
C04599=1182.827,27.215,-46.440,-179.670,5.863,148.946
C04600=1182.822,27.464,-46.455,-179.667,5.864,148.945
C04601=1182.818,27.714,-46.470,-179.664,5.864,148.945
C04602=1182.812,27.964,-46.485,-179.662,5.865,148.944
C04603=1182.807,28.232,-46.500,-179.660,5.866,148.944
C04604=1182.801,28.501,-46.517,-179.656,5.867,148.943
C04605=1182.796,28.770,-46.533,-179.654,5.868,148.942
C04606=1182.790,29.039,-46.549,-179.651,5.868,148.942
C04607=1182.786,29.288,-46.564,-179.649,5.869,148.941
C04608=1182.781,29.538,-46.579,-179.646,5.869,148.940
C04609=1182.775,29.787,-46.594,-179.643,5.871,148.940
C04610=1182.771,30.037,-46.608,-179.641,5.872,148.939
C04611=1182.765,30.286,-46.624,-179.638,5.872,148.939
C04612=1182.760,30.535,-46.639,-179.636,5.873,148.938
C04613=1182.756,30.786,-46.654,-179.633,5.873,148.938
C04614=1182.751,31.035,-46.669,-179.631,5.874,148.937
C04615=1182.746,31.284,-46.684,-179.628,5.874,148.936
C04616=1182.740,31.534,-46.699,-179.626,5.875,148.936
C04617=1182.736,31.783,-46.714,-179.623,5.877,148.935
C04618=1182.730,32.033,-46.730,-179.620,5.877,148.934
C04619=1182.726,32.282,-46.745,-179.618,5.878,148.934
C04620=1182.720,32.532,-46.760,-179.615,5.878,148.933
C04621=1182.715,32.781,-46.775,-179.613,5.879,148.933
C04622=1182.710,33.030,-46.790,-179.610,5.880,148.932
C04623=1182.706,33.281,-46.805,-179.608,5.880,148.931
C04624=1182.700,33.530,-46.820,-179.605,5.882,148.931
C04625=1182.696,33.779,-46.835,-179.602,5.883,148.930
C04626=1182.690,34.028,-46.851,-179.600,5.883,148.930
C04627=1182.686,34.278,-46.866,-179.597,5.884,148.929
C04628=1182.680,34.528,-46.881,-179.595,5.884,148.929
C04629=1182.675,34.777,-46.896,-179.592,5.885,148.928
C04630=1182.670,35.027,-46.912,-179.589,5.886,148.927
C04631=1182.666,35.276,-46.927,-179.587,5.887,148.927
C04632=1182.660,35.525,-46.942,-179.584,5.888,148.926
C04633=1182.655,35.775,-46.957,-179.582,5.888,148.926
C04634=1182.650,36.024,-46.972,-179.580,5.889,148.925
C04635=1182.645,36.274,-46.988,-179.577,5.889,148.924
C04636=1182.641,36.524,-47.003,-179.575,5.890,148.924
C04637=1182.635,36.773,-47.019,-179.571,5.892,148.923
C04638=1182.631,37.022,-47.034,-179.569,5.892,148.922
C04639=1182.625,37.271,-47.049,-179.567,5.893,148.922
C04640=1182.620,37.521,-47.065,-179.564,5.894,148.921
C04641=1182.615,37.771,-47.080,-179.561,5.894,148.921
C04642=1182.610,38.021,-47.095,-179.559,5.895,148.920
C04643=1182.605,38.270,-47.110,-179.556,5.896,148.920
C04644=1182.600,38.519,-47.126,-179.553,5.897,148.919
C04645=1182.595,38.769,-47.141,-179.551,5.898,148.918
C04646=1182.591,39.018,-47.157,-179.549,5.898,148.918
C04647=1182.585,39.268,-47.172,-179.546,5.899,148.917
C04648=1182.580,39.517,-47.188,-179.543,5.900,148.917
C04649=1182.575,39.766,-47.203,-179.541,5.901,148.916
C04650=1182.570,40.016,-47.218,-179.538,5.902,148.916
C04651=1182.565,40.266,-47.234,-179.536,5.902,148.915
C04652=1182.560,40.515,-47.249,-179.533,5.903,148.914
C04653=1182.555,40.764,-47.265,-179.531,5.904,148.914
C04654=1182.550,41.014,-47.281,-179.528,5.905,148.913
C04655=1182.546,41.263,-47.296,-179.525,5.905,148.912
C04656=1182.540,41.513,-47.312,-179.523,5.906,148.912
C04657=1182.535,41.762,-47.327,-179.520,5.907,148.911
C04658=1182.530,42.011,-47.342,-179.518,5.908,148.911
C04659=1182.525,42.261,-47.358,-179.515,5.909,148.910
C04660=1182.520,42.511,-47.374,-179.512,5.909,148.909
C04661=1182.515,42.760,-47.389,-179.510,5.910,148.909
C04662=1182.511,43.010,-47.405,-179.507,5.911,148.908
C04663=1182.505,43.259,-47.421,-179.505,5.911,148.908
C04664=1182.500,43.508,-47.437,-179.502,5.913,148.907
C04665=1182.495,43.758,-47.452,-179.499,5.914,148.907
C04666=1182.491,44.007,-47.467,-179.497,5.914,148.906
C04667=1182.485,44.257,-47.483,-179.495,5.915,148.905
C04668=1182.480,44.506,-47.499,-179.492,5.915,148.905
C04669=1182.475,44.756,-47.515,-179.489,5.917,148.904
C04670=1182.470,45.006,-47.530,-179.487,5.918,148.904
C04671=1182.465,45.254,-47.546,-179.484,5.918,148.903
C04672=1182.461,45.504,-47.562,-179.482,5.919,148.903
C04673=1182.455,45.754,-47.577,-179.479,5.920,148.902
C04674=1182.450,46.003,-47.593,-179.476,5.921,148.901
C04675=1182.445,46.253,-47.609,-179.474,5.922,148.901
C04676=1182.441,46.502,-47.625,-179.471,5.922,148.900
C04677=1182.435,46.751,-47.640,-179.469,5.923,148.900
C04678=1182.430,47.001,-47.656,-179.466,5.924,148.899
C04679=1182.425,47.251,-47.672,-179.464,5.925,148.899
C04680=1182.420,47.499,-47.688,-179.461,5.926,148.898
C04681=1182.415,47.750,-47.704,-179.458,5.926,148.897
C04682=1182.411,47.999,-47.719,-179.456,5.928,148.897
C04683=1182.405,48.248,-47.735,-179.453,5.929,148.896
C04684=1182.401,48.497,-47.751,-179.450,5.929,148.895
C04685=1182.395,48.747,-47.767,-179.448,5.930,148.895
C04686=1182.391,48.997,-47.783,-179.446,5.930,148.894
C04687=1182.385,49.246,-47.799,-179.443,5.932,148.894
C04688=1182.380,49.495,-47.815,-179.440,5.933,148.893
C04689=1182.375,49.745,-47.831,-179.438,5.933,148.893
C04690=1182.371,49.994,-47.846,-179.435,5.934,148.892
C04691=1182.366,50.244,-47.862,-179.432,5.935,148.891
C04692=1182.361,50.493,-47.878,-179.430,5.936,148.891
C04693=1182.356,50.742,-47.894,-179.427,5.937,148.890
C04694=1182.351,50.992,-47.910,-179.425,5.937,148.890
C04695=1182.345,51.242,-47.926,-179.422,5.939,148.889
C04696=1182.341,51.491,-47.942,-179.419,5.939,148.889
C04697=1182.336,51.740,-47.958,-179.417,5.940,148.888
C04698=1182.331,51.990,-47.975,-179.415,5.941,148.887
C04699=1182.326,52.239,-47.990,-179.411,5.942,148.887
C04700=1182.321,52.488,-48.007,-179.409,5.943,148.886
C04701=1182.316,52.738,-48.023,-179.407,5.944,148.886
C04702=1182.311,52.988,-48.038,-179.404,5.944,148.885
C04703=1182.306,53.237,-48.055,-179.401,5.946,148.885
C04704=1182.301,53.486,-48.070,-179.399,5.946,148.884
C04705=1182.296,53.736,-48.087,-179.396,5.947,148.883
C04706=1182.291,53.985,-48.103,-179.394,5.948,148.883
C04707=1182.286,54.253,-48.120,-179.391,5.949,148.882
C04708=1182.281,54.522,-48.138,-179.388,5.950,148.882
C04709=1182.275,54.791,-48.155,-179.385,5.951,148.881
C04710=1182.269,55.059,-48.172,-179.383,5.952,148.880
C04711=1182.265,55.309,-48.188,-179.380,5.953,148.880
C04712=1182.260,55.558,-48.205,-179.377,5.954,148.879
C04713=1182.255,55.808,-48.221,-179.375,5.954,148.879
C04714=1182.250,56.057,-48.237,-179.372,5.955,148.878
C04715=1182.244,56.307,-48.254,-179.369,5.957,148.877
C04716=1182.239,56.556,-48.270,-179.367,5.958,148.877
C04717=1182.235,56.806,-48.286,-179.364,5.958,148.876
C04718=1182.230,57.055,-48.302,-179.362,5.959,148.876
C04719=1182.225,57.304,-48.319,-179.359,5.960,148.875
C04720=1182.220,57.554,-48.334,-179.356,5.961,148.875
C04721=1182.215,57.803,-48.351,-179.354,5.962,148.874
C04722=1182.210,58.052,-48.367,-179.351,5.963,148.874
C04723=1182.205,58.302,-48.383,-179.349,5.964,148.873
C04724=1182.200,58.551,-48.400,-179.346,5.964,148.872
C04725=1182.195,58.801,-48.416,-179.344,5.965,148.872
C04726=1182.190,59.051,-48.433,-179.341,5.967,148.871
C04727=1182.185,59.299,-48.449,-179.338,5.967,148.871
C04728=1182.180,59.549,-48.465,-179.336,5.968,148.870
C04729=1182.175,59.798,-48.481,-179.333,5.969,148.870
C04730=1182.171,60.048,-48.498,-179.331,5.970,148.869
C04731=1182.165,60.297,-48.515,-179.328,5.971,148.868
C04732=1182.160,60.547,-48.531,-179.325,5.972,148.868
C04733=1182.155,60.796,-48.547,-179.323,5.973,148.867
C04734=1182.151,61.045,-48.564,-179.320,5.974,148.867
C04735=1182.146,61.295,-48.581,-179.318,5.974,148.866
C04736=1182.140,61.544,-48.597,-179.315,5.976,148.866
C04737=1182.136,61.794,-48.613,-179.313,5.977,148.865
C04738=1182.130,62.043,-48.630,-179.310,5.977,148.864
C04739=1182.126,62.292,-48.646,-179.307,5.979,148.864
C04740=1182.121,62.542,-48.662,-179.305,5.979,148.863
C04741=1182.115,62.791,-48.679,-179.302,5.980,148.863
C04742=1182.111,63.041,-48.696,-179.299,5.982,148.862
C04743=1182.106,63.290,-48.712,-179.297,5.982,148.862
C04744=1182.101,63.539,-48.729,-179.294,5.983,148.861
C04745=1182.096,63.789,-48.746,-179.291,5.984,148.861
C04746=1182.091,64.038,-48.762,-179.289,5.985,148.860
C04747=1182.086,64.288,-48.778,-179.286,5.986,148.859
C04748=1182.081,64.538,-48.796,-179.283,5.987,148.859
C04749=1182.076,64.786,-48.812,-179.281,5.988,148.858
C04750=1182.072,65.036,-48.829,-179.278,5.989,148.858
C04751=1182.067,65.285,-48.845,-179.276,5.990,148.857
C04752=1182.061,65.534,-48.862,-179.273,5.991,148.857
C04753=1182.057,65.784,-48.879,-179.271,5.992,148.856
C04754=1182.052,66.033,-48.896,-179.268,5.993,148.855
C04755=1182.046,66.282,-48.912,-179.266,5.994,148.855
C04756=1182.042,66.533,-48.928,-179.263,5.994,148.854
C04757=1182.037,66.782,-48.945,-179.260,5.996,148.854
C04758=1182.031,67.031,-48.962,-179.258,5.997,148.853
C04759=1182.027,67.281,-48.979,-179.255,5.997,148.853
C04760=1182.022,67.530,-48.995,-179.252,5.999,148.852
C04761=1182.017,67.779,-49.012,-179.250,5.999,148.852
C04762=1182.012,68.029,-49.029,-179.247,6.000,148.851
C04763=1182.008,68.278,-49.046,-179.244,6.002,148.850
C04764=1182.002,68.528,-49.063,-179.242,6.003,148.850
C04765=1181.997,68.777,-49.079,-179.239,6.003,148.849
C04766=1181.992,69.027,-49.096,-179.237,6.005,148.849
C04767=1181.988,69.275,-49.114,-179.234,6.005,148.848
C04768=1181.983,69.524,-49.130,-179.231,6.006,148.848
C04769=1181.978,69.774,-49.147,-179.229,6.008,148.847
C04770=1181.973,70.023,-49.164,-179.226,6.008,148.847
C04771=1181.968,70.273,-49.181,-179.223,6.010,148.846
C04772=1181.963,70.522,-49.198,-179.221,6.010,148.845
C04773=1181.958,70.772,-49.215,-179.219,6.011,148.845
C04774=1181.953,71.021,-49.232,-179.215,6.013,148.844
C04775=1181.949,71.271,-49.248,-179.213,6.013,148.844
C04776=1181.943,71.520,-49.265,-179.211,6.014,148.843
C04777=1181.939,71.769,-49.282,-179.208,6.016,148.843
C04778=1181.933,72.019,-49.300,-179.205,6.016,148.842
C04779=1181.929,72.268,-49.316,-179.203,6.018,148.842
C04780=1181.923,72.517,-49.333,-179.200,6.018,148.841
C04781=1181.919,72.767,-49.350,-179.198,6.019,148.841
C04782=1181.913,73.016,-49.367,-179.195,6.021,148.840
C04783=1181.909,73.265,-49.385,-179.192,6.022,148.840
C04784=1181.904,73.515,-49.402,-179.190,6.022,148.839
C04785=1181.899,73.764,-49.418,-179.187,6.024,148.838
C04786=1181.894,74.014,-49.435,-179.184,6.024,148.838
C04787=1181.890,74.263,-49.453,-179.182,6.026,148.837
C04788=1181.884,74.512,-49.470,-179.179,6.027,148.837
C04789=1181.879,74.762,-49.487,-179.176,6.027,148.836
C04790=1181.874,75.011,-49.504,-179.174,6.029,148.836
C04791=1181.869,75.260,-49.522,-179.171,6.029,148.835
C04792=1181.865,75.510,-49.538,-179.168,6.031,148.835
C04793=1181.859,75.759,-49.556,-179.166,6.032,148.834
C04794=1181.855,76.009,-49.572,-179.164,6.033,148.833
C04795=1181.850,76.258,-49.590,-179.160,6.034,148.833
C04796=1181.844,76.507,-49.607,-179.158,6.035,148.832
C04797=1181.840,76.757,-49.624,-179.155,6.036,148.832
C04798=1181.835,77.006,-49.642,-179.153,6.037,148.831
C04799=1181.830,77.255,-49.658,-179.150,6.038,148.831
C04800=1181.825,77.505,-49.676,-179.148,6.039,148.830
C04801=1181.820,77.754,-49.694,-179.145,6.040,148.830
C04802=1181.816,78.004,-49.710,-179.142,6.041,148.829
C04803=1181.810,78.252,-49.728,-179.140,6.042,148.829
C04804=1181.805,78.502,-49.745,-179.137,6.043,148.828
C04805=1181.801,78.751,-49.762,-179.134,6.044,148.827
C04806=1181.796,79.001,-49.780,-179.132,6.045,148.827
C04807=1181.790,79.250,-49.797,-179.129,6.047,148.826
C04808=1181.786,79.499,-49.815,-179.127,6.047,148.826
C04809=1181.781,79.749,-49.832,-179.124,6.049,148.825
C04810=1181.776,79.998,-49.850,-179.121,6.050,148.825
C04811=1181.771,80.266,-49.868,-179.118,6.051,148.824
C04812=1181.765,80.535,-49.886,-179.116,6.052,148.824
C04813=1181.760,80.803,-49.906,-179.113,6.053,148.823
C04814=1181.755,81.072,-49.924,-179.110,6.054,148.822
C04815=1181.751,81.321,-49.942,-179.107,6.056,148.822
C04816=1181.745,81.570,-49.959,-179.105,6.056,148.821
C04817=1181.740,81.819,-49.977,-179.102,6.058,148.821
C04818=1181.735,82.069,-49.994,-179.100,6.058,148.820
C04819=1181.731,82.318,-50.011,-179.097,6.060,148.820
C04820=1181.725,82.568,-50.028,-179.094,6.061,148.819
C04821=1181.721,82.817,-50.046,-179.092,6.061,148.819
C04822=1181.715,83.067,-50.064,-179.089,6.063,148.818
C04823=1181.711,83.316,-50.081,-179.087,6.064,148.818
C04824=1181.706,83.565,-50.099,-179.083,6.065,148.817
C04825=1181.701,83.815,-50.116,-179.081,6.066,148.817
C04826=1181.696,84.064,-50.134,-179.078,6.067,148.816
C04827=1181.691,84.313,-50.152,-179.076,6.068,148.816
C04828=1181.687,84.562,-50.169,-179.073,6.070,148.815
C04829=1181.682,84.812,-50.187,-179.071,6.070,148.815
C04830=1181.677,85.061,-50.204,-179.069,6.071,148.814
C04831=1181.672,85.311,-50.222,-179.065,6.073,148.813
C04832=1181.667,85.560,-50.240,-179.063,6.074,148.813
C04833=1181.662,85.809,-50.257,-179.060,6.075,148.812
C04834=1181.657,86.058,-50.275,-179.058,6.076,148.812
C04835=1181.653,86.308,-50.293,-179.055,6.077,148.811
C04836=1181.647,86.557,-50.310,-179.052,6.078,148.811
C04837=1181.642,86.806,-50.328,-179.049,6.080,148.810
C04838=1181.637,87.056,-50.346,-179.047,6.080,148.810
C04839=1181.633,87.305,-50.364,-179.044,6.082,148.809
C04840=1181.627,87.555,-50.381,-179.042,6.083,148.809
C04841=1181.622,87.804,-50.399,-179.039,6.084,148.808
C04842=1181.618,88.053,-50.417,-179.036,6.085,148.808
C04843=1181.613,88.302,-50.435,-179.034,6.087,148.807
C04844=1181.608,88.552,-50.452,-179.031,6.087,148.807
C04845=1181.603,88.801,-50.470,-179.029,6.088,148.806
C04846=1181.598,89.050,-50.488,-179.026,6.089,148.806
C04847=1181.593,89.299,-50.506,-179.024,6.090,148.805
C04848=1181.589,89.549,-50.524,-179.020,6.092,148.804
C04849=1181.584,89.799,-50.541,-179.018,6.093,148.804
C04850=1181.579,90.048,-50.559,-179.015,6.094,148.803
C04851=1181.574,90.297,-50.577,-179.013,6.095,148.803
C04852=1181.569,90.546,-50.595,-179.010,6.097,148.803
C04853=1181.564,90.796,-50.613,-179.008,6.097,148.802
C04854=1181.559,91.045,-50.631,-179.005,6.099,148.801
C04855=1181.554,91.294,-50.649,-179.002,6.099,148.801
C04856=1181.549,91.543,-50.667,-179.000,6.101,148.800
C04857=1181.545,91.792,-50.685,-178.997,6.102,148.800
C04858=1181.539,92.042,-50.703,-178.994,6.103,148.799
C04859=1181.535,92.292,-50.721,-178.992,6.104,148.799
C04860=1181.530,92.541,-50.739,-178.989,6.106,148.798
C04861=1181.525,92.790,-50.757,-178.987,6.107,148.798
C04862=1181.520,93.039,-50.775,-178.984,6.108,148.797
C04863=1181.515,93.289,-50.793,-178.981,6.109,148.797
C04864=1181.510,93.538,-50.811,-178.978,6.110,148.796
C04865=1181.506,93.787,-50.829,-178.976,6.111,148.796
C04866=1181.501,94.037,-50.847,-178.973,6.113,148.795
C04867=1181.496,94.286,-50.865,-178.971,6.113,148.795
C04868=1181.491,94.535,-50.883,-178.968,6.115,148.794
C04869=1181.487,94.784,-50.901,-178.965,6.116,148.794
C04870=1181.482,95.034,-50.919,-178.963,6.117,148.793
C04871=1181.477,95.283,-50.937,-178.960,6.118,148.793
C04872=1181.472,95.533,-50.956,-178.957,6.120,148.792
C04873=1181.467,95.782,-50.974,-178.954,6.121,148.792
C04874=1181.462,96.031,-50.993,-178.952,6.122,148.791
C04875=1181.457,96.280,-51.011,-178.949,6.124,148.791
C04876=1181.452,96.529,-51.029,-178.947,6.124,148.790
C04877=1181.447,96.778,-51.047,-178.944,6.126,148.790
C04878=1181.443,97.028,-51.065,-178.941,6.127,148.789
C04879=1181.437,97.278,-51.083,-178.939,6.128,148.789
C04880=1181.433,97.527,-51.101,-178.936,6.129,148.788
C04881=1181.428,97.776,-51.119,-178.933,6.131,148.787
C04882=1181.423,98.025,-51.137,-178.931,6.131,148.787
C04883=1181.419,98.274,-51.156,-178.928,6.133,148.786
C04884=1181.414,98.523,-51.174,-178.926,6.134,148.786
C04885=1181.408,98.773,-51.193,-178.923,6.135,148.786
C04886=1181.403,99.022,-51.211,-178.920,6.136,148.785
C04887=1181.399,99.272,-51.229,-178.918,6.138,148.785
C04888=1181.394,99.521,-51.248,-178.915,6.139,148.784
C04889=1181.389,99.770,-51.266,-178.912,6.140,148.783
C04890=1181.384,100.019,-51.285,-178.910,6.142,148.783
C04891=1181.379,100.269,-51.303,-178.907,6.142,148.782
C04892=1181.375,100.518,-51.322,-178.904,6.144,148.782
C04893=1181.370,100.767,-51.340,-178.902,6.145,148.781
C04894=1181.364,101.016,-51.358,-178.899,6.146,148.781
C04895=1181.360,101.266,-51.377,-178.897,6.147,148.781
C04896=1181.355,101.515,-51.395,-178.894,6.149,148.780
C04897=1181.350,101.764,-51.413,-178.891,6.150,148.780
C04898=1181.345,102.014,-51.432,-178.888,6.151,148.779
C04899=1181.341,102.263,-51.451,-178.886,6.153,148.778
C04900=1181.336,102.512,-51.469,-178.884,6.153,148.778
C04901=1181.330,102.761,-51.487,-178.880,6.155,148.777
C04902=1181.326,103.011,-51.506,-178.878,6.156,148.777
C04903=1181.321,103.260,-51.524,-178.875,6.157,148.776
C04904=1181.316,103.509,-51.542,-178.872,6.159,148.776
C04905=1181.312,103.759,-51.562,-178.870,6.160,148.776
C04906=1181.307,104.008,-51.580,-178.867,6.161,148.775
C04907=1181.302,104.256,-51.599,-178.865,6.162,148.774
C04908=1181.297,104.506,-51.618,-178.862,6.164,148.774
C04909=1181.292,104.756,-51.636,-178.860,6.164,148.773
C04910=1181.287,105.005,-51.655,-178.857,6.166,148.773
C04911=1181.282,105.254,-51.673,-178.854,6.167,148.772
C04912=1181.278,105.503,-51.692,-178.852,6.168,148.772
C04913=1181.272,105.752,-51.711,-178.849,6.170,148.772
C04914=1181.268,106.002,-51.730,-178.846,6.171,148.771
C04915=1181.262,106.270,-51.750,-178.843,6.172,148.770
C04916=1181.257,106.539,-51.769,-178.840,6.174,148.770
C04917=1181.252,106.807,-51.790,-178.838,6.175,148.769
C04918=1181.247,107.075,-51.810,-178.834,6.177,148.769
C04919=1181.242,107.324,-51.829,-178.832,6.178,148.768
C04920=1181.238,107.574,-51.847,-178.829,6.179,148.768
C04921=1181.232,107.823,-51.867,-178.827,6.180,148.767
C04922=1181.228,108.073,-51.885,-178.824,6.182,148.767
C04923=1181.223,108.322,-51.904,-178.821,6.183,148.766
C04924=1181.218,108.570,-51.923,-178.819,6.184,148.766
C04925=1181.214,108.820,-51.941,-178.816,6.186,148.766
C04926=1181.208,109.069,-51.960,-178.814,6.186,148.765
C04927=1181.204,109.319,-51.979,-178.811,6.188,148.764
C04928=1181.199,109.568,-51.998,-178.808,6.190,148.764
C04929=1181.194,109.816,-52.017,-178.806,6.190,148.763
C04930=1181.189,110.067,-52.036,-178.803,6.192,148.763
C04931=1181.184,110.315,-52.054,-178.801,6.193,148.763
C04932=1181.180,110.565,-52.074,-178.797,6.194,148.762
C04933=1181.175,110.814,-52.092,-178.795,6.196,148.762
C04934=1181.170,111.063,-52.112,-178.793,6.197,148.761
C04935=1181.165,111.312,-52.131,-178.789,6.198,148.761
C04936=1181.160,111.562,-52.149,-178.787,6.200,148.760
C04937=1181.155,111.811,-52.169,-178.785,6.201,148.760
C04938=1181.150,112.060,-52.187,-178.781,6.203,148.759
C04939=1181.145,112.310,-52.206,-178.779,6.203,148.759
C04940=1181.141,112.558,-52.225,-178.777,6.205,148.758
C04941=1181.136,112.808,-52.245,-178.773,6.207,148.758
C04942=1181.131,113.056,-52.263,-178.771,6.207,148.757
C04943=1181.126,113.307,-52.282,-178.769,6.209,148.757
C04944=1181.121,113.556,-52.302,-178.765,6.211,148.756
C04945=1181.117,113.805,-52.321,-178.763,6.211,148.756
C04946=1181.112,114.054,-52.340,-178.761,6.213,148.755
C04947=1181.107,114.303,-52.360,-178.757,6.215,148.755
C04948=1181.102,114.552,-52.378,-178.755,6.216,148.754
C04949=1181.097,114.802,-52.397,-178.753,6.217,148.754
C04950=1181.093,115.050,-52.416,-178.749,6.219,148.753
C04951=1181.088,115.300,-52.436,-178.747,6.220,148.753
C04952=1181.083,115.549,-52.455,-178.744,6.221,148.752
C04953=1181.079,115.798,-52.474,-178.742,6.222,148.752
C04954=1181.073,116.047,-52.493,-178.739,6.224,148.751
C04955=1181.068,116.297,-52.512,-178.736,6.225,148.751
C04956=1181.064,116.547,-52.531,-178.734,6.226,148.751
C04957=1181.059,116.795,-52.550,-178.731,6.228,148.750
C04958=1181.054,117.045,-52.570,-178.728,6.229,148.750
C04959=1181.049,117.294,-52.589,-178.726,6.230,148.749
C04960=1181.045,117.543,-52.609,-178.723,6.232,148.749
C04961=1181.039,117.792,-52.628,-178.720,6.233,148.748
C04962=1181.035,118.042,-52.647,-178.718,6.234,148.748
C04963=1181.030,118.290,-52.666,-178.715,6.236,148.747
C04964=1181.025,118.540,-52.686,-178.712,6.237,148.747
C04965=1181.021,118.789,-52.705,-178.710,6.238,148.746
C04966=1181.015,119.038,-52.725,-178.707,6.240,148.746
C04967=1181.011,119.287,-52.744,-178.704,6.242,148.745
C04968=1181.006,119.536,-52.763,-178.702,6.243,148.745
C04969=1181.001,119.786,-52.783,-178.700,6.244,148.744
C04970=1180.996,120.035,-52.802,-178.696,6.246,148.744
C04971=1180.991,120.284,-52.822,-178.694,6.247,148.743
C04972=1180.987,120.533,-52.841,-178.692,6.248,148.743
C04973=1180.982,120.782,-52.860,-178.688,6.250,148.742
C04974=1180.977,121.032,-52.880,-178.686,6.251,148.742
C04975=1180.972,121.281,-52.899,-178.684,6.252,148.742
C04976=1180.967,121.530,-52.919,-178.681,6.254,148.741
C04977=1180.963,121.779,-52.938,-178.678,6.255,148.741
C04978=1180.958,122.029,-52.958,-178.676,6.256,148.740
C04979=1180.953,122.277,-52.977,-178.673,6.258,148.740
C04980=1180.948,122.527,-52.997,-178.670,6.260,148.739
C04981=1180.944,122.777,-53.017,-178.668,6.260,148.739
C04982=1180.938,123.025,-53.036,-178.665,6.262,148.738
C04983=1180.934,123.275,-53.055,-178.662,6.264,148.738
C04984=1180.930,123.524,-53.075,-178.659,6.265,148.737
C04985=1180.925,123.772,-53.095,-178.657,6.266,148.737
C04986=1180.920,124.022,-53.114,-178.654,6.268,148.737
C04987=1180.915,124.272,-53.134,-178.651,6.270,148.736
C04988=1180.910,124.520,-53.154,-178.649,6.270,148.736
C04989=1180.905,124.769,-53.174,-178.646,6.272,148.735
C04990=1180.901,125.019,-53.193,-178.643,6.274,148.735
C04991=1180.896,125.269,-53.213,-178.641,6.275,148.734
C04992=1180.891,125.517,-53.233,-178.638,6.276,148.734
C04993=1180.886,125.766,-53.253,-178.635,6.278,148.733
C04994=1180.882,126.016,-53.272,-178.633,6.280,148.733
C04995=1180.877,126.264,-53.291,-178.631,6.280,148.733
C04996=1180.872,126.513,-53.311,-178.627,6.282,148.732
C04997=1180.867,126.763,-53.331,-178.625,6.284,148.731
C04998=1180.863,127.013,-53.351,-178.622,6.285,148.731
C04999=1180.858,127.261,-53.371,-178.620,6.286,148.731
C05000=1180.853,127.510,-53.390,-178.617,6.288,148.730
C05001=1180.848,127.760,-53.410,-178.614,6.289,148.730
C05002=1180.844,128.009,-53.430,-178.611,6.291,148.729
C05003=1180.838,128.258,-53.450,-178.609,6.292,148.729
C05004=1180.834,128.507,-53.470,-178.606,6.293,148.728
C05005=1180.829,128.756,-53.490,-178.603,6.295,148.728
C05006=1180.825,129.006,-53.509,-178.601,6.297,148.727
C05007=1180.819,129.254,-53.529,-178.598,6.298,148.727
C05008=1180.815,129.504,-53.549,-178.595,6.299,148.726
C05009=1180.810,129.753,-53.569,-178.593,6.301,148.726
C05010=1180.805,130.003,-53.590,-178.590,6.303,148.726
C05011=1180.800,130.251,-53.610,-178.588,6.304,148.725
C05012=1180.795,130.500,-53.629,-178.585,6.305,148.725
C05013=1180.791,130.749,-53.650,-178.582,6.307,148.724
C05014=1180.786,130.999,-53.669,-178.579,6.309,148.724
C05015=1180.781,131.248,-53.690,-178.577,6.310,148.723
C05016=1180.777,131.497,-53.709,-178.574,6.311,148.723
C05017=1180.772,131.746,-53.729,-178.571,6.313,148.722
C05018=1180.767,131.995,-53.749,-178.568,6.314,148.722
C05019=1180.762,132.264,-53.771,-178.566,6.316,148.722
C05020=1180.757,132.532,-53.793,-178.563,6.318,148.721
C05021=1180.751,132.801,-53.814,-178.560,6.319,148.721
C05022=1180.746,133.069,-53.836,-178.557,6.321,148.720
C05023=1180.742,133.319,-53.856,-178.555,6.322,148.720
C05024=1180.736,133.568,-53.877,-178.552,6.323,148.719
C05025=1180.732,133.818,-53.896,-178.549,6.325,148.719
C05026=1180.727,134.067,-53.917,-178.546,6.327,148.718
C05027=1180.723,134.315,-53.937,-178.544,6.328,148.718
C05028=1180.718,134.565,-53.957,-178.541,6.329,148.717
C05029=1180.712,134.814,-53.977,-178.538,6.331,148.717
C05030=1180.708,135.063,-53.998,-178.536,6.333,148.717
C05031=1180.703,135.312,-54.017,-178.533,6.334,148.716
C05032=1180.699,135.561,-54.038,-178.531,6.335,148.716
C05033=1180.694,135.810,-54.058,-178.528,6.337,148.715
C05034=1180.689,136.060,-54.078,-178.525,6.339,148.715
C05035=1180.684,136.309,-54.099,-178.522,6.340,148.715
C05036=1180.680,136.558,-54.119,-178.520,6.342,148.714
C05037=1180.675,136.807,-54.139,-178.518,6.343,148.714
C05038=1180.669,137.056,-54.159,-178.514,6.344,148.713
C05039=1180.665,137.305,-54.180,-178.512,6.346,148.713
C05040=1180.661,137.554,-54.200,-178.509,6.348,148.712
C05041=1180.655,137.803,-54.221,-178.506,6.350,148.712
C05042=1180.651,138.052,-54.241,-178.504,6.351,148.712
C05043=1180.646,138.302,-54.261,-178.501,6.352,148.711
C05044=1180.642,138.551,-54.281,-178.498,6.354,148.711
C05045=1180.637,138.800,-54.302,-178.496,6.356,148.710
C05046=1180.632,139.049,-54.323,-178.493,6.357,148.710
C05047=1180.628,139.298,-54.343,-178.491,6.358,148.709
C05048=1180.622,139.547,-54.364,-178.488,6.360,148.709
C05049=1180.618,139.797,-54.384,-178.485,6.362,148.709
C05050=1180.613,140.045,-54.404,-178.482,6.363,148.708
C05051=1180.608,140.295,-54.425,-178.480,6.365,148.708
C05052=1180.604,140.544,-54.445,-178.477,6.366,148.707
C05053=1180.599,140.793,-54.466,-178.475,6.368,148.707
C05054=1180.594,141.042,-54.487,-178.472,6.369,148.706
C05055=1180.590,141.291,-54.507,-178.469,6.371,148.706
C05056=1180.584,141.540,-54.528,-178.466,6.372,148.705
C05057=1180.580,141.789,-54.549,-178.463,6.374,148.705
C05058=1180.576,142.038,-54.569,-178.461,6.375,148.705
C05059=1180.570,142.287,-54.590,-178.459,6.377,148.704
C05060=1180.566,142.536,-54.610,-178.456,6.379,148.704
C05061=1180.561,142.785,-54.631,-178.453,6.380,148.703
C05062=1180.556,143.034,-54.652,-178.450,6.382,148.703
C05063=1180.551,143.284,-54.673,-178.447,6.384,148.703
C05064=1180.547,143.533,-54.693,-178.445,6.385,148.702
C05065=1180.542,143.782,-54.713,-178.443,6.386,148.702
C05066=1180.537,144.031,-54.734,-178.440,6.388,148.701
C05067=1180.533,144.280,-54.755,-178.437,6.390,148.701
C05068=1180.528,144.529,-54.776,-178.435,6.392,148.701
C05069=1180.523,144.778,-54.796,-178.431,6.393,148.700
C05070=1180.518,145.027,-54.817,-178.429,6.395,148.700
C05071=1180.513,145.276,-54.837,-178.427,6.396,148.699
C05072=1180.509,145.526,-54.859,-178.424,6.397,148.699
C05073=1180.504,145.775,-54.879,-178.421,6.399,148.698
C05074=1180.500,146.024,-54.901,-178.418,6.401,148.698
C05075=1180.495,146.273,-54.921,-178.416,6.403,148.698
C05076=1180.490,146.522,-54.942,-178.413,6.404,148.697
C05077=1180.486,146.771,-54.962,-178.410,6.406,148.697
C05078=1180.480,147.020,-54.983,-178.408,6.407,148.696
C05079=1180.475,147.269,-55.004,-178.405,6.409,148.696
C05080=1180.471,147.518,-55.025,-178.402,6.410,148.696
C05081=1180.466,147.767,-55.046,-178.400,6.412,148.695
C05082=1180.462,148.017,-55.067,-178.397,6.414,148.695
C05083=1180.457,148.266,-55.088,-178.394,6.416,148.694
C05084=1180.452,148.515,-55.108,-178.392,6.417,148.694
C05085=1180.448,148.763,-55.130,-178.389,6.418,148.693
C05086=1180.442,149.013,-55.151,-178.386,6.420,148.693
C05087=1180.438,149.262,-55.171,-178.384,6.421,148.693
C05088=1180.433,149.510,-55.193,-178.381,6.423,148.692
C05089=1180.429,149.760,-55.214,-178.378,6.425,148.692
C05090=1180.424,150.009,-55.235,-178.376,6.427,148.691
C05091=1180.419,150.259,-55.256,-178.373,6.428,148.691
C05092=1180.415,150.507,-55.277,-178.370,6.430,148.691
C05093=1180.410,150.756,-55.298,-178.368,6.432,148.690
C05094=1180.404,151.005,-55.319,-178.365,6.433,148.690
C05095=1180.400,151.255,-55.341,-178.362,6.434,148.689
C05096=1180.396,151.504,-55.361,-178.360,6.436,148.689
C05097=1180.391,151.752,-55.383,-178.357,6.438,148.689
C05098=1180.386,152.002,-55.404,-178.354,6.440,148.688
C05099=1180.381,152.250,-55.424,-178.351,6.441,148.688
C05100=1180.377,152.500,-55.446,-178.349,6.443,148.687
C05101=1180.372,152.749,-55.467,-178.346,6.445,148.687
C05102=1180.368,152.997,-55.488,-178.343,6.447,148.687
C05103=1180.363,153.247,-55.509,-178.341,6.448,148.686
C05104=1180.358,153.495,-55.531,-178.339,6.449,148.686
C05105=1180.353,153.745,-55.552,-178.336,6.451,148.686
C05106=1180.349,153.994,-55.573,-178.333,6.453,148.685
C05107=1180.344,154.243,-55.594,-178.330,6.454,148.685
C05108=1180.339,154.492,-55.615,-178.327,6.456,148.684
C05109=1180.334,154.741,-55.637,-178.325,6.458,148.684
C05110=1180.329,154.991,-55.658,-178.322,6.460,148.683
C05111=1180.325,155.239,-55.679,-178.319,6.461,148.683
C05112=1180.320,155.488,-55.701,-178.317,6.463,148.683
C05113=1180.316,155.738,-55.723,-178.314,6.465,148.682
C05114=1180.311,155.986,-55.744,-178.311,6.467,148.682
C05115=1180.306,156.236,-55.765,-178.309,6.468,148.682
C05116=1180.301,156.484,-55.786,-178.306,6.470,148.681
C05117=1180.297,156.734,-55.808,-178.304,6.471,148.681
C05118=1180.292,156.982,-55.829,-178.301,6.473,148.680
C05119=1180.287,157.231,-55.851,-178.298,6.475,148.680
C05120=1180.282,157.481,-55.872,-178.296,6.476,148.680
C05121=1180.278,157.730,-55.894,-178.293,6.478,148.679
C05122=1180.273,157.978,-55.916,-178.290,6.480,148.679
C05123=1180.268,158.247,-55.938,-178.287,6.481,148.678
C05124=1180.263,158.517,-55.962,-178.284,6.484,148.678
C05125=1180.258,158.786,-55.985,-178.281,6.486,148.678
C05126=1180.253,159.055,-56.009,-178.279,6.487,148.677
C05127=1180.247,159.304,-56.030,-178.276,6.489,148.677
C05128=1180.244,159.553,-56.051,-178.273,6.491,148.676
C05129=1180.239,159.802,-56.073,-178.271,6.493,148.676
C05130=1180.234,160.050,-56.094,-178.267,6.494,148.676
C05131=1180.230,160.300,-56.116,-178.265,6.496,148.675
C05132=1180.225,160.549,-56.137,-178.262,6.498,148.675
C05133=1180.220,160.797,-56.159,-178.259,6.500,148.674
C05134=1180.216,161.047,-56.181,-178.257,6.501,148.674
C05135=1180.210,161.296,-56.202,-178.254,6.503,148.674
C05136=1180.206,161.545,-56.224,-178.252,6.504,148.673
C05137=1180.201,161.794,-56.246,-178.249,6.506,148.673
C05138=1180.196,162.043,-56.268,-178.246,6.508,148.673
C05139=1180.192,162.292,-56.290,-178.244,6.509,148.672
C05140=1180.187,162.541,-56.311,-178.241,6.511,148.672
C05141=1180.182,162.789,-56.333,-178.238,6.513,148.671
C05142=1180.178,163.039,-56.354,-178.236,6.515,148.671
C05143=1180.173,163.288,-56.376,-178.233,6.516,148.671
C05144=1180.169,163.537,-56.398,-178.230,6.518,148.670
C05145=1180.164,163.786,-56.420,-178.228,6.520,148.670
C05146=1180.159,164.034,-56.441,-178.225,6.522,148.670
C05147=1180.155,164.284,-56.463,-178.222,6.523,148.669
C05148=1180.150,164.532,-56.485,-178.220,6.525,148.669
C05149=1180.146,164.782,-56.507,-178.217,6.527,148.668
C05150=1180.141,165.030,-56.529,-178.214,6.529,148.668
C05151=1180.136,165.280,-56.551,-178.212,6.531,148.668
C05152=1180.131,165.529,-56.573,-178.209,6.532,148.667
C05153=1180.127,165.778,-56.595,-178.206,6.534,148.667
C05154=1180.122,166.027,-56.617,-178.204,6.536,148.667
C05155=1180.117,166.276,-56.639,-178.201,6.538,148.666
C05156=1180.113,166.525,-56.661,-178.198,6.539,148.666
C05157=1180.108,166.773,-56.682,-178.195,6.541,148.665
C05158=1180.103,167.023,-56.704,-178.193,6.543,148.665
C05159=1180.098,167.272,-56.727,-178.190,6.545,148.665
C05160=1180.094,167.521,-56.749,-178.187,6.546,148.664
C05161=1180.089,167.770,-56.770,-178.185,6.548,148.664
C05162=1180.084,168.019,-56.792,-178.182,6.550,148.664
C05163=1180.080,168.268,-56.814,-178.179,6.552,148.663
C05164=1180.075,168.517,-56.836,-178.177,6.554,148.663
C05165=1180.070,168.765,-56.859,-178.174,6.555,148.663
C05166=1180.066,169.015,-56.881,-178.171,6.557,148.662
C05167=1180.061,169.263,-56.903,-178.169,6.559,148.662
C05168=1180.057,169.513,-56.925,-178.166,6.561,148.661
C05169=1180.051,169.762,-56.947,-178.163,6.562,148.661
C05170=1180.047,170.011,-56.969,-178.161,6.564,148.661
C05171=1180.043,170.260,-56.992,-178.158,6.566,148.660
C05172=1180.038,170.508,-57.014,-178.156,6.568,148.660
C05173=1180.033,170.758,-57.036,-178.153,6.570,148.660
C05174=1180.028,171.007,-57.058,-178.150,6.572,148.659
C05175=1180.024,171.256,-57.080,-178.148,6.573,148.659
C05176=1180.019,171.504,-57.102,-178.144,6.576,148.659
C05177=1180.014,171.754,-57.125,-178.142,6.578,148.658
C05178=1180.009,172.002,-57.147,-178.139,6.580,148.658
C05179=1180.005,172.252,-57.169,-178.136,6.581,148.658
C05180=1180.000,172.501,-57.192,-178.134,6.583,148.657
C05181=1179.995,172.749,-57.214,-178.131,6.585,148.657
C05182=1179.991,172.999,-57.236,-178.128,6.587,148.657
C05183=1179.986,173.247,-57.259,-178.126,6.588,148.656
C05184=1179.982,173.496,-57.281,-178.123,6.590,148.656
C05185=1179.977,173.746,-57.303,-178.120,6.592,148.655
C05186=1179.972,173.994,-57.326,-178.118,6.594,148.655
C05187=1179.968,174.243,-57.348,-178.115,6.595,148.655
C05188=1179.963,174.491,-57.370,-178.112,6.597,148.654
C05189=1179.958,174.741,-57.393,-178.110,6.599,148.654
C05190=1179.954,174.990,-57.415,-178.107,6.601,148.654
C05191=1179.949,175.238,-57.438,-178.105,6.603,148.654
C05192=1179.944,175.488,-57.460,-178.102,6.605,148.653
C05193=1179.940,175.737,-57.483,-178.099,6.606,148.653
C05194=1179.935,175.986,-57.505,-178.097,6.608,148.652
C05195=1179.931,176.234,-57.528,-178.093,6.611,148.652
C05196=1179.926,176.484,-57.551,-178.091,6.613,148.652
C05197=1179.921,176.732,-57.573,-178.088,6.614,148.651
C05198=1179.917,176.981,-57.595,-178.085,6.616,148.651
C05199=1179.912,177.230,-57.618,-178.083,6.618,148.651
C05200=1179.907,177.479,-57.640,-178.080,6.620,148.650
C05201=1179.903,177.728,-57.663,-178.077,6.622,148.650
C05202=1179.898,177.977,-57.685,-178.075,6.623,148.650
C05203=1179.893,178.226,-57.708,-178.073,6.625,148.649
C05204=1179.889,178.475,-57.731,-178.070,6.627,148.649
C05205=1179.884,178.724,-57.754,-178.067,6.629,148.649
C05206=1179.879,178.973,-57.776,-178.065,6.631,148.648
C05207=1179.875,179.222,-57.799,-178.062,6.633,148.648
C05208=1179.871,179.470,-57.822,-178.059,6.635,148.648
C05209=1179.866,179.720,-57.844,-178.056,6.637,148.647
C05210=1179.861,179.968,-57.867,-178.053,6.639,148.647
C05211=1179.856,180.217,-57.890,-178.051,6.640,148.647
C05212=1179.852,180.466,-57.912,-178.048,6.642,148.646
C05213=1179.847,180.716,-57.936,-178.046,6.644,148.646
C05214=1179.843,180.964,-57.958,-178.043,6.646,148.646
C05215=1179.838,181.213,-57.981,-178.040,6.648,148.645
C05216=1179.833,181.462,-58.004,-178.038,6.650,148.645
C05217=1179.829,181.711,-58.027,-178.035,6.651,148.645
C05218=1179.824,181.960,-58.049,-178.032,6.654,148.644
C05219=1179.820,182.209,-58.072,-178.029,6.656,148.644
C05220=1179.815,182.458,-58.095,-178.026,6.658,148.644
C05221=1179.810,182.707,-58.118,-178.024,6.660,148.643
C05222=1179.805,182.955,-58.140,-178.022,6.662,148.643
C05223=1179.801,183.204,-58.163,-178.019,6.663,148.643
C05224=1179.797,183.453,-58.186,-178.016,6.665,148.642
C05225=1179.792,183.702,-58.210,-178.014,6.667,148.642
C05226=1179.787,183.951,-58.233,-178.010,6.669,148.642
C05227=1179.783,184.221,-58.257,-178.008,6.671,148.641
C05228=1179.777,184.490,-58.282,-178.005,6.673,148.641
C05229=1179.772,184.760,-58.307,-178.002,6.676,148.641
C05230=1179.767,185.030,-58.332,-177.999,6.677,148.640
C05231=1179.763,185.279,-58.355,-177.996,6.679,148.640
C05232=1179.757,185.527,-58.378,-177.994,6.681,148.640
C05233=1179.753,185.776,-58.401,-177.991,6.683,148.639
C05234=1179.749,186.025,-58.424,-177.988,6.686,148.639
C05235=1179.744,186.274,-58.447,-177.986,6.688,148.639
C05236=1179.739,186.523,-58.470,-177.983,6.689,148.638
C05237=1179.735,186.772,-58.493,-177.980,6.691,148.638
C05238=1179.730,187.020,-58.516,-177.978,6.693,148.638
C05239=1179.725,187.269,-58.539,-177.975,6.695,148.637
C05240=1179.720,187.518,-58.563,-177.973,6.697,148.637
C05241=1179.716,187.767,-58.586,-177.969,6.699,148.637
C05242=1179.712,188.016,-58.609,-177.967,6.701,148.636
C05243=1179.707,188.265,-58.632,-177.964,6.703,148.636
C05244=1179.702,188.514,-58.656,-177.961,6.705,148.636
C05245=1179.698,188.763,-58.679,-177.959,6.707,148.635
C05246=1179.693,189.011,-58.701,-177.957,6.709,148.635
C05247=1179.688,189.260,-58.725,-177.953,6.711,148.635
C05248=1179.684,189.509,-58.748,-177.951,6.713,148.635
C05249=1179.679,189.758,-58.772,-177.948,6.715,148.634
C05250=1179.675,190.007,-58.796,-177.945,6.717,148.634
C05251=1179.670,190.256,-58.819,-177.943,6.718,148.634
C05252=1179.666,190.505,-58.842,-177.940,6.721,148.633
C05253=1179.661,190.754,-58.865,-177.937,6.723,148.633
C05254=1179.657,191.003,-58.888,-177.934,6.725,148.633
C05255=1179.652,191.252,-58.912,-177.932,6.727,148.632
C05256=1179.647,191.501,-58.935,-177.929,6.728,148.632
C05257=1179.643,191.749,-58.959,-177.927,6.731,148.632
C05258=1179.638,191.998,-58.983,-177.924,6.732,148.632
C05259=1179.633,192.247,-59.006,-177.921,6.735,148.631
C05260=1179.629,192.496,-59.029,-177.918,6.737,148.631
C05261=1179.623,192.745,-59.052,-177.916,6.739,148.631
C05262=1179.620,192.993,-59.076,-177.914,6.741,148.630
C05263=1179.615,193.242,-59.099,-177.911,6.742,148.630
C05264=1179.610,193.491,-59.123,-177.908,6.744,148.630
C05265=1179.606,193.740,-59.146,-177.905,6.747,148.629
C05266=1179.601,193.988,-59.170,-177.902,6.749,148.629
C05267=1179.597,194.237,-59.193,-177.900,6.751,148.629
C05268=1179.592,194.486,-59.217,-177.897,6.753,148.629
C05269=1179.587,194.735,-59.240,-177.895,6.754,148.628
C05270=1179.583,194.984,-59.264,-177.892,6.757,148.628
C05271=1179.578,195.233,-59.287,-177.889,6.759,148.628
C05272=1179.573,195.482,-59.311,-177.887,6.761,148.627
C05273=1179.570,195.731,-59.335,-177.884,6.763,148.627
C05274=1179.565,195.980,-59.359,-177.881,6.764,148.627
C05275=1179.560,196.228,-59.383,-177.878,6.767,148.626
C05276=1179.556,196.477,-59.406,-177.876,6.769,148.626
C05277=1179.551,196.726,-59.429,-177.873,6.771,148.626
C05278=1179.546,196.975,-59.454,-177.871,6.773,148.626
C05279=1179.541,197.224,-59.477,-177.867,6.775,148.625
C05280=1179.537,197.473,-59.501,-177.865,6.778,148.625
C05281=1179.532,197.722,-59.525,-177.862,6.779,148.625
C05282=1179.528,197.970,-59.549,-177.860,6.781,148.624
C05283=1179.523,198.219,-59.572,-177.857,6.783,148.624
C05284=1179.519,198.467,-59.596,-177.854,6.786,148.624
C05285=1179.514,198.716,-59.620,-177.852,6.788,148.624
C05286=1179.510,198.965,-59.644,-177.849,6.789,148.623
C05287=1179.505,199.214,-59.667,-177.846,6.791,148.623
C05288=1179.500,199.463,-59.692,-177.843,6.794,148.623
C05289=1179.496,199.712,-59.716,-177.841,6.796,148.622
C05290=1179.491,199.961,-59.740,-177.838,6.798,148.622
C05291=1179.486,200.210,-59.763,-177.836,6.800,148.622
C05292=1179.482,200.458,-59.787,-177.833,6.802,148.622
C05293=1179.477,200.707,-59.810,-177.830,6.804,148.621
C05294=1179.473,200.956,-59.834,-177.828,6.806,148.621
C05295=1179.468,201.204,-59.859,-177.825,6.808,148.621
C05296=1179.464,201.454,-59.883,-177.823,6.810,148.620
C05297=1179.459,201.703,-59.907,-177.819,6.813,148.620
C05298=1179.455,201.951,-59.931,-177.817,6.814,148.620
C05299=1179.450,202.200,-59.954,-177.814,6.816,148.619
C05300=1179.445,202.449,-59.979,-177.812,6.818,148.619
C05301=1179.441,202.697,-60.003,-177.809,6.821,148.619
C05302=1179.437,202.947,-60.027,-177.806,6.823,148.619
C05303=1179.432,203.195,-60.051,-177.803,6.825,148.618
C05304=1179.427,203.444,-60.076,-177.801,6.827,148.618
C05305=1179.422,203.693,-60.099,-177.798,6.829,148.618
C05306=1179.418,203.941,-60.123,-177.795,6.831,148.618
C05307=1179.414,204.190,-60.147,-177.793,6.833,148.617
C05308=1179.409,204.439,-60.172,-177.790,6.836,148.617
C05309=1179.404,204.688,-60.196,-177.787,6.838,148.617
C05310=1179.400,204.937,-60.220,-177.784,6.839,148.616
C05311=1179.395,205.185,-60.244,-177.782,6.842,148.616
C05312=1179.391,205.435,-60.269,-177.779,6.844,148.616
C05313=1179.387,205.683,-60.293,-177.776,6.846,148.616
C05314=1179.381,205.932,-60.317,-177.774,6.848,148.616
C05315=1179.377,206.181,-60.341,-177.772,6.850,148.615
C05316=1179.372,206.429,-60.365,-177.768,6.852,148.615
C05317=1179.368,206.679,-60.390,-177.766,6.855,148.615
C05318=1179.364,206.927,-60.414,-177.763,6.856,148.614
C05319=1179.358,207.176,-60.439,-177.760,6.859,148.614
C05320=1179.354,207.424,-60.463,-177.758,6.861,148.614
C05321=1179.350,207.673,-60.487,-177.755,6.863,148.614
C05322=1179.345,207.922,-60.512,-177.753,6.865,148.613
C05323=1179.341,208.170,-60.536,-177.749,6.867,148.613
C05324=1179.335,208.420,-60.560,-177.747,6.869,148.613
C05325=1179.331,208.669,-60.584,-177.745,6.871,148.613
C05326=1179.327,208.917,-60.608,-177.741,6.874,148.612
C05327=1179.322,209.166,-60.633,-177.739,6.876,148.612
C05328=1179.318,209.415,-60.657,-177.737,6.878,148.612
C05329=1179.313,209.664,-60.682,-177.733,6.880,148.611
C05330=1179.309,209.912,-60.706,-177.731,6.883,148.611
C05331=1179.304,210.183,-60.733,-177.728,6.884,148.611
C05332=1179.299,210.453,-60.760,-177.725,6.887,148.611
C05333=1179.294,210.723,-60.787,-177.722,6.890,148.610
C05334=1179.289,210.994,-60.813,-177.719,6.891,148.610
C05335=1179.285,211.243,-60.838,-177.717,6.894,148.610
C05336=1179.280,211.491,-60.863,-177.714,6.896,148.610
C05337=1179.275,211.740,-60.887,-177.712,6.898,148.609
C05338=1179.271,211.989,-60.912,-177.709,6.900,148.609
C05339=1179.266,212.238,-60.936,-177.706,6.903,148.609
C05340=1179.262,212.487,-60.961,-177.704,6.905,148.609
C05341=1179.257,212.735,-60.986,-177.701,6.907,148.608
C05342=1179.253,212.984,-61.010,-177.698,6.909,148.608
C05343=1179.248,213.233,-61.035,-177.696,6.911,148.608
C05344=1179.244,213.481,-61.059,-177.693,6.913,148.608
C05345=1179.239,213.730,-61.084,-177.690,6.916,148.607
C05346=1179.234,213.979,-61.110,-177.688,6.918,148.607
C05347=1179.230,214.227,-61.134,-177.685,6.920,148.607
C05348=1179.225,214.477,-61.159,-177.682,6.922,148.607
C05349=1179.221,214.725,-61.183,-177.679,6.925,148.606
C05350=1179.216,214.973,-61.208,-177.677,6.926,148.606
C05351=1179.212,215.223,-61.233,-177.674,6.929,148.606
C05352=1179.207,215.471,-61.257,-177.671,6.931,148.606
C05353=1179.203,215.721,-61.282,-177.669,6.933,148.605
C05354=1179.198,215.969,-61.308,-177.666,6.936,148.605
C05355=1179.194,216.218,-61.332,-177.663,6.938,148.605
C05356=1179.189,216.467,-61.357,-177.661,6.939,148.605
C05357=1179.184,216.715,-61.382,-177.658,6.942,148.604
C05358=1179.180,216.964,-61.407,-177.655,6.944,148.604
C05359=1179.176,217.212,-61.432,-177.652,6.947,148.604
C05360=1179.171,217.461,-61.457,-177.650,6.949,148.604
C05361=1179.167,217.710,-61.481,-177.647,6.951,148.603
C05362=1179.162,217.959,-61.507,-177.644,6.954,148.603
C05363=1179.157,218.207,-61.532,-177.642,6.955,148.603
C05364=1179.154,218.456,-61.557,-177.640,6.958,148.603
C05365=1179.149,218.704,-61.582,-177.636,6.960,148.603
C05366=1179.144,218.954,-61.607,-177.634,6.962,148.602
C05367=1179.139,219.202,-61.632,-177.632,6.964,148.602
C05368=1179.136,219.451,-61.656,-177.628,6.967,148.602
C05369=1179.131,219.699,-61.682,-177.626,6.969,148.602
C05370=1179.126,219.949,-61.707,-177.623,6.972,148.601
C05371=1179.121,220.197,-61.732,-177.620,6.973,148.601
C05372=1179.117,220.446,-61.757,-177.618,6.976,148.601
C05373=1179.113,220.694,-61.782,-177.615,6.978,148.601
C05374=1179.108,220.943,-61.808,-177.613,6.980,148.600
C05375=1179.103,221.191,-61.832,-177.610,6.982,148.600
C05376=1179.099,221.440,-61.858,-177.607,6.985,148.600
C05377=1179.094,221.689,-61.883,-177.605,6.987,148.600
C05378=1179.090,221.938,-61.909,-177.601,6.989,148.599
C05379=1179.085,222.186,-61.933,-177.599,6.992,148.599
C05380=1179.081,222.435,-61.958,-177.597,6.993,148.599
C05381=1179.077,222.684,-61.984,-177.594,6.996,148.599
C05382=1179.072,222.933,-62.009,-177.591,6.998,148.599
C05383=1179.068,223.181,-62.035,-177.588,7.001,148.598
C05384=1179.063,223.429,-62.060,-177.586,7.003,148.598
C05385=1179.058,223.679,-62.085,-177.583,7.005,148.598
C05386=1179.053,223.927,-62.110,-177.580,7.008,148.598
C05387=1179.049,224.176,-62.136,-177.578,7.010,148.597
C05388=1179.046,224.424,-62.161,-177.575,7.012,148.597
C05389=1179.041,224.673,-62.186,-177.572,7.014,148.597
C05390=1179.036,224.922,-62.212,-177.570,7.016,148.597
C05391=1179.031,225.170,-62.237,-177.567,7.019,148.597
C05392=1179.027,225.419,-62.263,-177.565,7.021,148.596
C05393=1179.023,225.668,-62.288,-177.561,7.024,148.596
C05394=1179.018,225.916,-62.313,-177.559,7.026,148.596
C05395=1179.014,226.165,-62.339,-177.557,7.028,148.596
C05396=1179.009,226.414,-62.365,-177.554,7.031,148.596
C05397=1179.005,226.662,-62.390,-177.551,7.033,148.595
C05398=1179.000,226.911,-62.415,-177.548,7.035,148.595
C05399=1178.995,227.160,-62.441,-177.546,7.037,148.595
C05400=1178.991,227.408,-62.466,-177.543,7.040,148.595
C05401=1178.987,227.657,-62.492,-177.540,7.042,148.595
C05402=1178.982,227.905,-62.517,-177.538,7.044,148.594
C05403=1178.978,228.154,-62.543,-177.535,7.047,148.594
C05404=1178.974,228.403,-62.569,-177.532,7.049,148.594
C05405=1178.969,228.651,-62.594,-177.530,7.052,148.594
C05406=1178.964,228.900,-62.620,-177.527,7.053,148.593
C05407=1178.959,229.149,-62.646,-177.524,7.056,148.593
C05408=1178.954,229.398,-62.671,-177.522,7.058,148.593
C05409=1178.950,229.646,-62.697,-177.519,7.060,148.593
C05410=1178.946,229.895,-62.723,-177.516,7.063,148.593
C05411=1178.942,230.144,-62.748,-177.514,7.065,148.592
C05412=1178.937,230.392,-62.774,-177.511,7.068,148.592
C05413=1178.933,230.641,-62.800,-177.509,7.070,148.592
C05414=1178.928,230.890,-62.825,-177.506,7.073,148.592
C05415=1178.924,231.137,-62.851,-177.503,7.075,148.592
C05416=1178.919,231.386,-62.878,-177.500,7.078,148.592
C05417=1178.915,231.635,-62.903,-177.498,7.079,148.591
C05418=1178.911,231.884,-62.929,-177.496,7.082,148.591
C05419=1178.906,232.132,-62.955,-177.492,7.084,148.591
C05420=1178.901,232.381,-62.980,-177.490,7.086,148.591
C05421=1178.897,232.630,-63.007,-177.487,7.089,148.590
C05422=1178.892,232.879,-63.032,-177.485,7.091,148.590
C05423=1178.887,233.127,-63.058,-177.482,7.094,148.590
C05424=1178.883,233.376,-63.084,-177.479,7.096,148.590
C05425=1178.879,233.624,-63.110,-177.476,7.099,148.590
C05426=1178.874,233.873,-63.136,-177.474,7.101,148.590
C05427=1178.870,234.122,-63.162,-177.471,7.103,148.589
C05428=1178.865,234.370,-63.188,-177.469,7.105,148.589
C05429=1178.861,234.619,-63.213,-177.466,7.108,148.589
C05430=1178.856,234.867,-63.240,-177.463,7.110,148.589
C05431=1178.852,235.116,-63.266,-177.460,7.113,148.589
C05432=1178.848,235.365,-63.292,-177.458,7.115,148.588
C05433=1178.843,235.613,-63.317,-177.456,7.117,148.588
C05434=1178.838,235.861,-63.344,-177.452,7.120,148.588
C05435=1178.834,236.133,-63.372,-177.450,7.123,148.588
C05436=1178.829,236.405,-63.401,-177.446,7.125,148.588
C05437=1178.824,236.677,-63.430,-177.444,7.128,148.588
C05438=1178.820,236.948,-63.459,-177.441,7.130,148.587
C05439=1178.815,237.196,-63.484,-177.438,7.133,148.587
C05440=1178.810,237.445,-63.510,-177.436,7.135,148.587
C05441=1178.806,237.693,-63.537,-177.433,7.138,148.587
C05442=1178.802,237.942,-63.562,-177.431,7.140,148.587
C05443=1178.797,238.191,-63.590,-177.427,7.143,148.586
C05444=1178.793,238.440,-63.615,-177.425,7.145,148.586
C05445=1178.789,238.688,-63.641,-177.422,7.147,148.586
C05446=1178.784,238.937,-63.668,-177.420,7.150,148.586
C05447=1178.779,239.185,-63.693,-177.417,7.153,148.586
C05448=1178.774,239.433,-63.721,-177.415,7.154,148.585
C05449=1178.770,239.682,-63.746,-177.412,7.157,148.585
C05450=1178.766,239.931,-63.773,-177.409,7.159,148.585
C05451=1178.761,240.180,-63.799,-177.406,7.162,148.585
C05452=1178.757,240.428,-63.826,-177.404,7.164,148.585
C05453=1178.752,240.677,-63.852,-177.401,7.167,148.585
C05454=1178.749,240.925,-63.878,-177.399,7.169,148.585
C05455=1178.744,241.174,-63.905,-177.396,7.172,148.584
C05456=1178.740,241.422,-63.931,-177.393,7.174,148.584
C05457=1178.735,241.671,-63.958,-177.391,7.177,148.584
C05458=1178.730,241.919,-63.984,-177.388,7.179,148.584
C05459=1178.725,242.168,-64.010,-177.385,7.182,148.584
C05460=1178.721,242.416,-64.036,-177.383,7.185,148.584
C05461=1178.717,242.665,-64.063,-177.380,7.186,148.583
C05462=1178.712,242.914,-64.089,-177.377,7.189,148.583
C05463=1178.708,243.162,-64.116,-177.375,7.191,148.583
C05464=1178.704,243.410,-64.143,-177.372,7.194,148.583
C05465=1178.699,243.659,-64.169,-177.370,7.196,148.583
C05466=1178.694,243.908,-64.196,-177.367,7.199,148.583
C05467=1178.690,244.156,-64.223,-177.364,7.201,148.582
C05468=1178.685,244.405,-64.249,-177.361,7.204,148.582
C05469=1178.681,244.653,-64.275,-177.359,7.206,148.582
C05470=1178.677,244.902,-64.303,-177.356,7.209,148.582
C05471=1178.673,245.150,-64.329,-177.354,7.211,148.582
C05472=1178.668,245.399,-64.355,-177.351,7.214,148.582
C05473=1178.663,245.648,-64.382,-177.348,7.217,148.581
C05474=1178.659,245.896,-64.409,-177.346,7.219,148.581
C05475=1178.655,246.144,-64.436,-177.343,7.222,148.581
C05476=1178.650,246.393,-64.462,-177.340,7.223,148.581
C05477=1178.646,246.642,-64.489,-177.338,7.226,148.581
C05478=1178.641,246.890,-64.516,-177.335,7.229,148.581
C05479=1178.637,247.138,-64.542,-177.332,7.231,148.581
C05480=1178.633,247.387,-64.570,-177.329,7.234,148.580
C05481=1178.628,247.636,-64.597,-177.327,7.236,148.580
C05482=1178.623,247.885,-64.623,-177.324,7.239,148.580
C05483=1178.620,248.133,-64.650,-177.322,7.241,148.580
C05484=1178.615,248.382,-64.677,-177.319,7.244,148.580
C05485=1178.610,248.630,-64.704,-177.317,7.246,148.580
C05486=1178.606,248.878,-64.730,-177.314,7.249,148.580
